IF MODE = 3 THEN
	z := 0;
	FOR n := 0 TO 4 DO (* konvertiere DWORD auf BYTE-Array *)
		FOR n1 := 0 TO 3 DO
			hash[n] := ROL(hash[n],8);
			SHA1[z] := DWORD_TO_BYTE(hash[n]);
			z := z + 1;
		END_FOR;
	END_FOR;
END_IF;

(* revision history

ks	6. dec. 2009 rev 1.0
	original version

*)

END_FUNCTION_BLOCK

// POUs/DATA_LOG/DLOG_STORE_RRD
FUNCTION_BLOCK DLOG_STORE_RRD
VAR_IN_OUT
	X : DLOG_DATA;
END_VAR
VAR_INPUT
	ENABLE : BOOL;
	TRIG_M : BOOL;
	TRIG_T : TIME;
	URL : STRING(OSCAT_BASIC.STRING_LENGTH);
	DTI : DT;
	SEP : BYTE;
	DNS_IP4 : DWORD;
	TIMEOUT : TIME;
END_VAR
VAR_OUTPUT
	ERROR_C : DWORD;
	ERROR_T : BYTE;
END_VAR
VAR
	UCB : UNI_CIRCULAR_BUFFER;
	IP_C : IP_C; (* IP_Control Verwaltungsstruktur *)
	S_BUF : NETWORK_BUFFER;
	R_BUF : NETWORK_BUFFER;
	URL_DATA : url;
	DNS_CLIENT : DNS_CLIENT;
	HTTP_GET : HTTP_GET;
	IPC : IP_CONTROL_V2;

	trig_auto : BOOL;
	trig_stored : BOOL;
	trig_tmp : BOOL;
	trig_m_last : BOOL;
	dti_last : DT := DT#2070-02-06-06:28:15;
	step_1 : INT;
	step_2 : INT;
	sep_char : STRING(1);
	url_query : STRING(OSCAT_BASIC.STRING_LENGTH);
	n : INT;

	(*
	LOG_MSG : LOG_MSG;
	_debug_enable : BOOL := TRUE;
	*)
END_VAR

(*
version 1.3		16. apr. 2012
programmer		ks
tested by			ks

DLOG_STORE_RRD der Baustein übergibt die DLOG Parameter an einen RoundRobinDatabase-Server
*)

X.DTI := DTI; (* Datum / Zeit eintragen *)
X.CLOCK_TRIG := DTI <> dti_last;
dti_last := DTI;
trig_auto := FALSE;
IF X.CLOCK_TRIG THEN (* Impuls in jeder Sekunde *)
	IF TRIG_T >= T#1000ms THEN (* automatischer Trigger *)
		trig_auto := DT_TO_UDINT(DTI) MOD (TIME_TO_UDINT(TRIG_T) / UDINT#1000) = UDINT#0;
	END_IF;
END_IF;

CASE step_1 OF

00:	IF ENABLE THEN
		X.ID_MAX := USINT#00;
		X.ADD_COM := 01; (* ADD INFO *)
		X.STORE_TYPE := BYTE#1; (* RRD-Modus *)

		ERROR_T := BYTE#0;
		ERROR_C := DWORD#0;

		X.UCB.D_MODE := 99;
		UCB(DATA:=X.UCB); (* Buffer löschen *)

		URL_DATA:=STRING_TO_URL(STR:=URL,DEFAULT_PROTOCOL:='',DEFAULT_PATH:=''); (* URL zerlegen *)
		sep_char := OSCAT_BASIC.CHR_TO_STRING(SEP);
		url_query := URL_DATA.QUERY;
		step_1 := 30;

		(* ---------------- Debug-Message -----------------------*)
		(*IF _debug_enable THEN
			LOG_CL.NEW_MSG := 'FILE_RRD1 - Start: DATE [~2]';
			LOG_CL.PRINTF[2] := DT_TO_STRING(DTI);
			LOG_MSG();
		END_IF;*)
		(* -----------------------------------------------------------------*)

	END_IF;

30:	(* LOG-Trigger verarbeiten *)
	trig_tmp := (TRIG_M AND NOT trig_m_last) OR trig_auto OR X.ADD_DATA_REQ;

	IF ENABLE = FALSE THEN (* ENABLE = 0 -> Log Stop *)
		X.ADD_COM := 00;
		step_1 := 00;

		(* ---------------- Debug-Message -----------------------*)
		(*IF _debug_enable THEN
			LOG_CL.NEW_MSG := 'FILE_RRD1 - Stop: DATE [~2]';
			LOG_CL.PRINTF[2] := DT_TO_STRING(DTI);
			LOG_MSG();
		END_IF;*)
		(* -----------------------------------------------------------------*)

	ELSIF ENABLE THEN
		IF trig_tmp OR trig_stored THEN (* manueller, automatischer oder externer Trigger *)
			trig_stored := FALSE;
			X.ADD_COM := 03; (* ADD DATA *)
			(* ---------------- Debug-Message -----------------------*)
			(*IF _debug_enable THEN
				LOG_CL.NEW_MSG := 'FILE_RRD1 - Trig: DATE [~2]';
				LOG_CL.PRINTF[2] := DT_TO_STRING(DTI);
				LOG_MSG();
			END_IF;*)
			(* -----------------------------------------------------------------*)
		ELSE
			X.ADD_COM := 04;	(* ADD DATA REQ *)
		END_IF;
	END_IF;

END_CASE;
X.ADD_DATA_REQ := FALSE; (* externe Anforderung rücksetzen *)

(* ##################################### *)

CASE step_2 OF

00:	IF X.UCB.BUF_COUNT >= USINT_TO_INT(X.ID_MAX) THEN (* genug Einträge vorhanden *)
		URL_DATA.QUERY := url_query; (* original Query wiederherstellen *)
		n := 1;
		WHILE n <= USINT_TO_INT(X.ID_MAX) DO
			X.UCB.D_MODE := 12; (* Element lesen und löschen *)
			UCB(DATA:=X.UCB);
			IF n < USINT_TO_INT(X.ID_MAX) THEN (* Trennzeichen hinzufügen *)
				X.UCB.D_STRING := CONCAT(X.UCB.D_STRING,sep_char);
			END_IF;
			IF LEN(X.UCB.D_STRING) + LEN(URL_DATA.QUERY) <= OSCAT_BASIC.STRING_LENGTH THEN
				URL_DATA.QUERY := CONCAT(URL_DATA.QUERY,X.UCB.D_STRING); (* Query mit LOG-Daten ergänzen *)
				step_2 := 40;
			ELSE
				ERROR_T := BYTE#4; (* LOG-Daten können nicht in URL gepackt werden *)
				ERROR_C := DWORD#1;
				step_2 := 100;
			END_IF;
			n := n + 1;
		END_WHILE;;
	END_IF;

40:	IF DNS_CLIENT.DONE THEN
		step_2 := 60;
	ELSIF (DNS_CLIENT.ERROR > DWORD#0) THEN
		ERROR_C := DNS_CLIENT.ERROR; (* Fehlerbehandlung *)
		ERROR_T := BYTE#1;
		step_2 := 100;
	END_IF;

60:	IF HTTP_GET.DONE THEN
		n := UINT_TO_INT(HTTP_GET.BODY_START);
		IF R_BUF.BUFFER[n] <> BYTE#48 THEN (* ASCII '0' *)
			ERROR_C := DWORD#1;
			ERROR_T := BYTE#3;
		END_IF;
		step_2 := 100;

	ELSIF HTTP_GET.ERROR > DWORD#0 THEN (* Fehlerbehandlung *)
		ERROR_C := HTTP_GET.ERROR;
		ERROR_T := BYTE#2;
		step_2 := 100;
	END_IF;

100:	IF (NOT HTTP_GET.DONE) THEN (* UNLOCK HTTP DATA *)
		step_2 := SEL(ERROR_T = BYTE#0, 120,0);
	END_IF;

120:	IF NOT ENABLE THEN
		step_2 := 0;
	END_IF;

END_CASE;

HTTP_GET(IP_C:=IP_C,S_BUF:=S_BUF,R_BUF:=R_BUF,IP4:=DNS_CLIENT.IP4,GET:=step_2=60,MODE:=2,UNLOCK_BUF:=step_2=100,URL_DATA:=URL_DATA); (* HTTP_GET *)
DNS_CLIENT(IP_C:=IP_C, S_BUF:=S_BUF, R_BUF:=R_BUF, DOMAIN:=URL_DATA.DOMAIN, IP4_DNS:= DNS_IP4, ACTIVATE:=step_2=40); (* DNS-Client *)
IPC(IP:= 0, PORT:= 0 , TIME_OUT:= TIMEOUT, IP_C:= IP_C, S_BUF:= S_BUF, R_BUF:= R_BUF); (* IP_CONTROL *)

trig_m_last := TRIG_M;

(* revision history
ks	01. jan. 2011	rev 1.0
	original version

ks	13. may. 2011	rev 1.1
	ADD_DATA_REQ hinzugefügt

ks	26. july. 2011	rev 1.2
	code optimierung D_MODE 12 und bessere fehlerauswertung

ks	16. apr. 2012	rev 1.3
	neuer überarbeiteter Code
*)

END_FUNCTION_BLOCK

// POUs/NETWORK/HTTP_GET
FUNCTION_BLOCK HTTP_GET
VAR_IN_OUT
	URL_DATA : url;
	IP_C : IP_C; (* IP_Control Verwaltungsstruktur *)
	S_BUF : NETWORK_BUFFER;
	R_BUF : NETWORK_BUFFER;
END_VAR
VAR_INPUT
	IP4 : DWORD;
	GET : BOOL;
	MODE : BYTE := BYTE#2;
	UNLOCK_BUF : BOOL;
END_VAR
VAR_OUTPUT
	HTTP_STATUS : STRING;
	HEADER_START : UINT; (* HTTP Header (Message Header) *)
	HEADER_STOP : UINT; (* HTTP Header (Message Header) *)
	BODY_START : UINT; (* Message Body *)
	BODY_STOP : UINT; (* Message Body *)
	DONE : BOOL;
	ERROR : DWORD;
END_VAR
VAR
	READ_HTTP :	READ_HTTP;
	IP_FIFO : IP_FIFO;
	ip_state : BYTE;
	ip_id : BYTE;
	get_last : BOOL;
	ip4_stored : DWORD;
	state : INT;
	i : INT;
	http_1_1_host : BOOL;
	total_size : INT;
	text : STRING(OSCAT_BASIC.STRING_LENGTH);
	delimiter2b : STRING(2);
	delimiter4b : STRING(4);
	del_end : STRING(4);
	del_pos : INT;
	idx : INT;
	rcv_timeout : BOOL;
	con_rdce : BOOL;

	(*LOG_MSG : LOG_MSG;
	_debug_enable : BOOL := TRUE;*)

END_VAR

(*

version 1.3	12. apr. 2011
programmer 	ks
tested by		ks

HTTP_GET führt eine HTTP Abfrage einer Web-Seite bei einem WEB_Server durch, und stellt die Daten ausbereitet zu verfügung
*)

CASE state OF
00:	IF GET AND NOT GET_LAST THEN (* auf positive Flanke SET warten *)
		state := 10;
		ip4_stored := IP4; (* aktuelle IP4 speichern *)
		DONE := FALSE;
		total_size := 0;
		HEADER_START := UINT#0;
		HEADER_STOP := UINT#0;
		BODY_START := UINT#0;
		BODY_STOP := UINT#0;
		HTTP_STATUS := '';
		ERROR := DWORD#0;
		ip_state := BYTE#1; (* Anmelden *)
		delimiter2b := '$0D$0A';
		delimiter4b := '$0D$0A$0D$0A';
	        	(*####################  DEBUG-MESSAGE  ###################################*)
		(*IF _debug_enable THEN
	       		LOG_CL.NEW_MSG := 'HTTP: S00 START /IP_ID ~4';
	            	LOG_CL.PRINTF[4]  := BYTE_TO_STRING(IP_ID);
	            	LOG_MSG();
	        	END_IF;*)
	        	(*########################################################################*)
	END_IF;

10:	IF ip_state = BYTE#3 THEN (* Bei IP_Control anmelden und auf freigabe warten *)
		idx := 0;
		text := CONCAT('GET ',URL_DATA.PATH);
		OSCAT_BASIC._STRING_TO_BUFFER(STR:=text,POS:=idx,PT:=ADR(S_BUF.BUFFER),SIZE:=SIZEOF(S_BUF.BUFFER)); (* GET path in buffer kopieren *)
		idx := idx + LEN(text);

		IF LEN(URL_DATA.QUERY) > 0 THEN
			S_BUF.BUFFER[idx] := 63; (* ASCII '?' *)
			idx := idx + 1;
			OSCAT_BASIC._STRING_TO_BUFFER(STR:=URL_DATA.QUERY,POS:=idx,PT:=ADR(S_BUF.BUFFER),SIZE:=SIZEOF(S_BUF.BUFFER)); (* QUERY in buffer kopieren *)
			idx := idx + LEN(URL_DATA.QUERY);
		END_IF;

		IF MODE >= BYTE#2 THEN (* gewünschte HTTP Version uebergeben *)
			text := ' HTTP/1.1';
		ELSE
			text := ' HTTP/1.0';
		END_IF;
		text := CONCAT(text,delimiter2b);
		OSCAT_BASIC._STRING_TO_BUFFER(STR:=text,POS:=idx,PT:=ADR(S_BUF.BUFFER),SIZE:=SIZEOF(S_BUF.BUFFER)); (* HTTP Version in buffer kopieren *)
		idx := idx + LEN(text);

		IF MODE = BYTE#1 THEN (* HTTP/1.0 mit persistenter Verbindung gewünscht *)
			text := CONCAT('Connection: Keep-Alive',delimiter2b); (* workaround für pcworx -> kein $0D$0A als Stringkonstante möglich *)
		ELSIF MODE = BYTE#3 THEN (* HTTP/1.1 ohne persistenter Verbindung gewünscht *)
			text := CONCAT('Connection: Close',delimiter2b); (* workaround für pcworx -> kein $0D$0A als Stringkonstante möglich *)
		ELSE
			text := '';
		END_IF;
		text := CONCAT(text,URL_DATA.HEADER);
		OSCAT_BASIC._STRING_TO_BUFFER(STR:=text,POS:=idx,PT:=ADR(S_BUF.BUFFER),SIZE:=SIZEOF(S_BUF.BUFFER)); (* HTTP Version in buffer kopieren *)
		idx := idx + LEN(text);

		text := CONCAT('Host: ',URL_DATA.DOMAIN);
		text := CONCAT(text,delimiter4b); (* workaround für pcworx -> kein $0D$0A als Stringkonstante möglich *)
		OSCAT_BASIC._STRING_TO_BUFFER(STR:=text,POS:=idx,PT:=ADR(S_BUF.BUFFER),SIZE:=SIZEOF(S_BUF.BUFFER)); (* HTTP Host in buffer kopieren *)
		idx := idx + LEN(text);

		(* IP Datenverkehr einrichten *)
		IF URL_DATA.PORT = WORD#0 THEN
			IP_C.C_PORT := WORD#80; (* Standard-Portnummer verwenden *)
		ELSE
			IP_C.C_PORT := URL_DATA.PORT; (* Portnummer aus URL verwenden *)
		END_IF;

		IP_C.C_IP := ip4_stored; (* IP eintragen *)
		IP_C.C_MODE := BYTE#0; (* Mode: TCP+AKTIV+PORT+IP *)
		IP_C.C_ENABLE := TRUE; (* Verbindungsaufbau freigeben *)
		IP_C.TIME_RESET := TRUE; (* Zeitueberwachung rücksetzen *)
		IP_C.R_OBSERVE := TRUE; (* Datenempfang ueberwachen *)
		S_BUF.SIZE := INT_TO_UINT(idx); (* Sendelänge eintragen *)
		R_BUF.SIZE := UINT#0; (* Empfangslänge rücksetzen *)

		state := 30;
	        	(*####################  DEBUG-MESSAGE  ###################################*)
	        	(*IF _debug_enable THEN
	        		LOG_CL.NEW_MSG := 'HTTP: S20 SEND /IP_ID ~4';
	            	LOG_CL.PRINTF[4]  := BYTE_TO_STRING(IP_ID);
	            	LOG_MSG();
	        	END_IF;*)
	        	(*########################################################################*)
	END_IF;

30:	rcv_timeout := (IP_C.ERROR AND DWORD#16#0000_FF00) = DWORD#16#0000_FF00;
	con_rdce :=     (IP_C.ERROR AND DWORD#16#FD00_0000) = DWORD#16#FD00_0000;

	IF S_BUF.SIZE = UINT#0 THEN
		IF total_size = 0 THEN
			IF R_BUF.SIZE > UINT#15 THEN; (* länge der empfangenen Daten prüfen *)

				(* HTTP HEADER Ende suchen -> durch $0D$A$0D$A erkennbar bei DEC RT-11,CP/M,MS-DOS,Windows *)
				del_end := '$0D$0A$0D$0A';
				del_pos := OSCAT_BASIC.BUFFER_SEARCH(PT:=ADR(R_BUF.BUFFER),SIZE:=R_BUF.SIZE,STR:=del_end,POS:=0,IGN:=FALSE);

				(* kein Ende gefunden ? -> andere Ende-Codierung suchen *)
				IF del_pos = 0 THEN
					del_end := '$0A$0A';
					(* HTTP HEADER Ende suchen -> durch $0A$0A erkennbar bei Multics, Unix-Derivate,Mac OS X *)
					del_pos := OSCAT_BASIC.BUFFER_SEARCH(PT:=ADR(R_BUF.BUFFER),SIZE:=R_BUF.SIZE,STR:=del_end,POS:=0,IGN:=FALSE);
				END_IF;

				IF del_pos > 0 THEN
					HEADER_START := UINT#0;
					HEADER_STOP := INT_TO_UINT(del_pos + LEN(del_end) - 1);
					TOTAL_SIZE := -1; (* HTTP Header empfangen aber noch keine gesamtlänge bekannt *)
				END_IF;
		                	(*####################  DEBUG-MESSAGE  ###################################*)
		                	(*IF _debug_enable THEN
		                   	LOG_CL.NEW_MSG := 'HTTP: S20 HEADER_START ~1 / HEADER_STOP ~2/IP_ID ~4';
		                   	LOG_CL.PRINTF[4]  := BYTE_TO_STRING(IP_ID);
		                   	LOG_CL.PRINTF[1]  := UINT_TO_STRING(HEADER_START);
		                   	LOG_CL.PRINTF[2]  := UINT_TO_STRING(HEADER_STOP);
		                   	LOG_MSG();
		                	END_IF;*)
		                	(*########################################################################*)

				(* HTTP Statuscode auswerten: (kann 1.0 oder 1.1 sein *)
				READ_HTTP(size:=HEADER_STOP,pos:=0,SRC:='',pt:=R_BUF.BUFFER);

				i := LEN(READ_HTTP.READ_HTTP);
				IF i > 7 THEN
					(* HTTP Version von HOST auswerten 1.0 oder 1.1 *)
					text:=MID(READ_HTTP.READ_HTTP,1,3);
					http_1_1_host := text = '1';

					(* Code und Meldung isolieren *)
					HTTP_STATUS := RIGHT(READ_HTTP.READ_HTTP,i-4);
				END_IF;

				(* positive HTTP Anfrage ? *)
				IF FIND(HTTP_STATUS,'200') > 0 THEN

					(* 'Content-Length: Wert einlesen auswerten *)
					READ_HTTP(size:=HEADER_STOP,pos:=0,SRC:='CONTENT-LENGTH',pt:=R_BUF.BUFFER);
					text:=READ_HTTP.READ_HTTP;

					IF LEN(text) >= 1 THEN
						IF OSCAT_BASIC.IS_NUM(str:=text) THEN
							(* erwartete gesamtmenge an Bytes berechnen *)
							total_size := STRING_TO_INT(text) + UINT_TO_INT(HEADER_STOP) + 1;
                           					(*####################  DEBUG-MESSAGE  ###################################*)
                           					(*IF _debug_enable THEN
                              					LOG_CL.NEW_MSG := 'HTTP: S20 HEADER ~1, BODY ~2 TOTAL ~3 /IP_ID ~4';
                             					LOG_CL.PRINTF[4]  := BYTE_TO_STRING(IP_ID);
                               					LOG_CL.PRINTF[1]  := UINT_TO_STRING(HEADER_STOP);
                               					LOG_CL.PRINTF[2]  := INT_TO_STRING(TOTAL_SIZE-UINT_TO_INT(HEADER_STOP));
                               					LOG_CL.PRINTF[3]  := INT_TO_STRING(TOTAL_SIZE);
                              					LOG_MSG();
                          					END_IF;*)
                          					(*########################################################################*)
						END_IF;
					END_IF;
				ELSE
					ERROR := DWORD#16#000000FC; (* Fehler durch HTTP-Statuscodes *)
				END_IF;
			END_IF;
		(* 1. bei bekannter Content-Length wird nach erhalt der erwartenen Daten die verbindung beendet *)
		(* 2. bei persistenter Verbindung muss bei unbekannter Datenmenge auf Receive-Timeout gewartet werden *)
		(* 3. wenn nach datenempfang die verbindung vom host unterbrochen wird *)
		ELSIF (R_BUF.SIZE >= INT_TO_UINT(total_size)) OR
			(R_BUF.SIZE > UINT#0 AND total_size < 0 AND ((rcv_timeout OR con_rdce) OR (IP_C.C_STATE = BYTE#1))) THEN

			IF R_BUF.SIZE - 1 > HEADER_STOP THEN (* BODY Daten vorhanden *)
				BODY_START := HEADER_STOP + UINT#1;
				BODY_STOP := R_BUF.SIZE - 1;
		                	(*####################  DEBUG-MESSAGE  ###################################*)
		                	(*IF _debug_enable THEN
		                   	LOG_CL.NEW_MSG := 'HTTP: S20 BODY ~1, START ~2 END ~3 /IP_ID ~4';
		                   	LOG_CL.PRINTF[4]  := BYTE_TO_STRING(IP_ID);
		                   	LOG_CL.PRINTF[1]  := UINT_TO_STRING(HEADER_STOP);
		                   	LOG_CL.PRINTF[2]  := UINT_TO_STRING(BODY_START);
		                   	LOG_CL.PRINTF[3]  := UINT_TO_STRING(BODY_STOP);
		                   	LOG_MSG();
		               	END_IF;*)
		               	(*########################################################################*)
			END_IF;

			DONE := TRUE;
			IP_C.C_ENABLE := FALSE; (* Verbindung abbauen *)
			state := 40;
            		(*####################  DEBUG-MESSAGE  ###################################*)
            		(*IF _debug_enable THEN
                			LOG_CL.NEW_MSG := 'HTTP: S30 OK /IP_ID ~4';
                			LOG_CL.PRINTF[4]  := BYTE_TO_STRING(IP_ID);
                			LOG_MSG();
            		END_IF;*)
            		(*########################################################################*)
		END_IF;
	END_IF;

	IF IP_C.ERROR <> DWORD#0 THEN
		(* bei unbekannter Content-size ist nicht bekannt ob bzw wieviele Telegramme noch folgen werden *)
		(* darum wird nach receive-timeout oder Remote disconnect error der fehler wieder ausgefiltert (logischer fehler) *)
		IF rcv_timeout AND DONE THEN
			IP_C.ERROR := IP_C.ERROR AND DWORD#16#FFFF_00FF; (* Fehler wieder rücksetzen *)
		ELSIF con_rdce AND DONE THEN
			IP_C.ERROR := IP_C.ERROR AND DWORD#16#00FF_FFFF; (* Fehler wieder rücksetzen *)
		ELSE
			ERROR := IP_C.ERROR;
		END_IF;
	END_IF;

	IF ERROR > DWORD#0 THEN
		IP_C.C_ENABLE := FALSE; (* Verbindungsaufbau sperren *)
		state := 40;
	        	(*####################  DEBUG-MESSAGE  ###################################*)
	        	(*IF _debug_enable THEN
	            	LOG_CL.NEW_MSG := 'HTTP: S30 ERROR ~1 /IP_ID ~4';
	            	LOG_CL.PRINTF[1]  := DWORD_TO_STRING(ERROR);
	            	LOG_CL.PRINTF[4]  := BYTE_TO_STRING(IP_ID);
	            	LOG_MSG();
	        	END_IF;*)
	        	(*########################################################################*)
	END_IF;

40:	IF (UNLOCK_BUF OR NOT DONE) THEN (* Warten auf Release und Verbindung beendet -> IP_ID vom Stack nehmen *)
		IP_STATE := BYTE#4; (* Abmelden *)
		DONE := FALSE;
		state := 0;
	END_IF;
END_CASE;

get_last := GET; (* letzten Status sichern zur Flankenerkennung *)

IP_FIFO(FIFO:=IP_C.FIFO,STATE:=ip_state,ID:=ip_id); (* IP_FIFO *)

(* revision history
ks	18. oct. 2008	rev 1.0
	original version

ks	20. oct. 2009	rev 1.1
	Fehler bei body-suche bei $0a$0a korrigiert,Codeoptimierung,
	new VAR del_pos , del_end (Networkbuffer und Buffer-funktionen auf Basis 0)

ks	28. oct. 2009	rev 1.2
	über url.header können zusätzliche header-infos übergeben werden

ks	12. apr. 2011	rev 1.3
	verbesserte fehlererkennung und fehlerkorrektur bei buffer_to_string
*)

END_FUNCTION_BLOCK

// POUs/NETWORK/READ_HTTP
FUNCTION_BLOCK READ_HTTP
VAR_INPUT
	SIZE : UINT;
	POS : INT;
	SRC : STRING;
END_VAR
VAR_IN_OUT
	PT : NW_BUF_LONG;
END_VAR
VAR_OUTPUT
	READ_HTTP : STRING(OSCAT_BASIC.STRING_LENGTH);
END_VAR
VAR
	index : INT;
	s1 : INT;
	e1 : INT;
	stop : INT;
END_VAR

(*

version 1.1 20. oct. 2009
programmer 	ks
tested by	ks

READ_HTTP wertet die Informationen einer HTTP-Request aus, und stellt die Daten zu Verfügung.
*)

stop := UINT_TO_INT(SIZE) - 1;

IF LEN(SRC) = 0 THEN
	(* wenn kein Suchbegriff vorhanden ist, dann den HTTP-STATUS auswerten *)
	SRC := 'HTTP/'; (* neuer Suchbegriff *)
ELSE
	(* gesuchten Parametertext ergänzen *)
	SRC := CONCAT(SRC,': ');
END_IF;

s1 := OSCAT_BASIC.BUFFER_SEARCH(pt:=ADR(PT),SIZE:=SIZE,STR:=SRC,POS:=POS,IGN:=TRUE);

IF s1 >= 0 THEN (* Text found *)
	e1 := s1;

	(* search start of line *)
	index := s1 - 1;
	WHILE (index > 0) DO
		IF pt[index] < BYTE#32 THEN EXIT; END_IF;
		s1 := s1 - 1;
		index := index - 1;
	END_WHILE;

	(* search end of line *)
	index := e1 + 1;
	WHILE (index <= stop) DO
		IF pt[index] < BYTE#32 THEN EXIT; END_IF;
		e1 := e1 + 1;
		index := index + 1;
	END_WHILE;

	s1 := s1 + LEN(SRC); (* 'suchbegriff: ' nicht mitkopieren *)

	(* copy string *)
	READ_HTTP := OSCAT_BASIC.BUFFER_TO_STRING(PT:=ADR(PT),SIZE:=SIZE,START:=s1,STOP:=e1);
ELSE
	READ_HTTP := '';
END_IF;

(* revision history

ks	18. oct. 2008	rev 1.0
	original version

ks	20. oct. 2009	rev 1.1
	Networkbuffer und Buffer-funktionen auf Basis 0

*)

END_FUNCTION_BLOCK

// POUs/DATA_LOG/DLOG_STRING
FUNCTION_BLOCK DLOG_STRING
VAR_IN_OUT
	X : DLOG_DATA;
END_VAR
VAR_INPUT
	STR : STRING;
	COLUMN : STRING(40);
END_VAR
VAR_OUTPUT
END_VAR
VAR
	UCB : UNI_CIRCULAR_BUFFER;
	id : WORD;
	str_last : STRING;
END_VAR

(*
version 1.3		19. apr. 2012
programmer		ks
tested by		ks

DLOG_STRING legt den STRING im FIFO-RING-Buffer ab um diesen mit den Baustein DLOG_STORE_*  aufzuzeichnen
*)

CASE x.ADD_COM OF

01:	(* ADD INFO *)
	X.ID_MAX := X.ID_MAX + USINT#1;
	id := WORD#16#0101; (* Quelltype STRING , Zieltype STRING *)
02:	(* ADD HEADER *)
	X.UCB.D_STRING := COLUMN;
	X.UCB.D_HEAD := id;
	X.UCB.D_MODE := 1;
	UCB(DATA:=X.UCB); (* Daten eintragen *)
03:	(* ADD DATA *)
	X.UCB.D_STRING := str_last;
	X.UCB.D_HEAD := id;
	X.UCB.D_MODE := 1;
	UCB(DATA:=X.UCB); (* Daten eintragen *)
END_CASE;
str_last := STR;

(* revision history
ks	01. jan. 2011	rev 1.0
	original version

ks	17. may. 2011	rev 1.1
	COLUMN STRING(40)

ks	25. july.   2011	rev 1.2
	neue head information

ks	19. apr.   2012	rev 1.3
	code neu überarbeitet
*)

END_FUNCTION_BLOCK

// POUs/NETWORK/DNS_DYN
FUNCTION_BLOCK DNS_DYN
VAR_IN_OUT
	IP_C : IP_C; (* IP_Control Verwaltungsstruktur *)
	S_BUF : NETWORK_BUFFER;
	R_BUF : NETWORK_BUFFER;
END_VAR
VAR_INPUT
	ENABLE : BOOL;
	UPDATE : BOOL;
	T_UPDATE : TIME := T#1h;
	MODE : BYTE;
	HOSTNAME : STRING(30);
	USERNAME : STRING(20);
	PASSWORD : STRING(20);
	IP4 : DWORD;
END_VAR
VAR_OUTPUT
	BUSY : BOOL;
	DONE : BOOL;
	ERROR_C : DWORD;
	ERROR_T : BYTE;
END_VAR
VAR
	DNS_CLIENT : DNS_CLIENT;
	HTTP_GET : HTTP_GET;
	BASE64_ENCODE_STR : BASE64_ENCODE_STR;
	URL_DATA : url;
	update_last : BOOL;
	state : INT;
	base64_done : BOOL;
	s1 : STRING(144);
	s2 : STRING(192);
	w : TON;
END_VAR

(*

version 1.2		02. dec. 2009
programmer 		ks
tested by		ks

YAHOO_WEATHER lädt vom Yahoo-Webserver einen Wetter RSS-Feed und analysiert die Daten und legt diese in einem Array ab
*)

CASE state OF

00:	IF ENABLE AND ((UPDATE AND NOT update_last) OR w.Q) THEN
		state := 20;
		DONE := FALSE;
		BUSY := TRUE;
		ERROR_C := DWORD#0;
		ERROR_T := BYTE#0;

		IF MODE = 0 THEN (* dyndns.org *)
			s2 := CONCAT('http://members.dyndns.org/nic/update?hostname=',HOSTNAME);
		ELSE (* selfhost.de *)
			s2 := 'http://carol.selfhost.de/nic/update?hostname=1';
		END_IF;
		IF IP4 > 0 THEN (* parametrierte IP verwenden *)
			s1 := CONCAT('&myip=',IP4_TO_STRING(IP4));
			s2 := CONCAT(s2,s1);
		END_IF;
		URL_DATA:=STRING_TO_URL(STR:=s2, DEFAULT_PROTOCOL:='', DEFAULT_PATH:=''); (* URL for DNS UND HTTP-GET *)
		s1 := CONCAT(USERNAME,':');
		s1 := CONCAT(s1,PASSWORD); (* BASE64 Encode Text *)
	END_IF;

20:	IF DNS_CLIENT.DONE THEN (* DNS_CLIENT *)
			state := 40;
	ELSIF (DNS_CLIENT.ERROR > DWORD#00) THEN (* Fehlerbehandlung *)
		ERROR_C := DNS_CLIENT.ERROR;
		ERROR_T := BYTE#01;
		BUSY := FALSE;
		state := 0;
	END_IF;

40: IF base64_done THEN (* BASE64 Encode beendet ? *)
		s1 := CONCAT('Authorization: Basic ',s2);
		s1 := CONCAT(s1,'$0D$0AUser-Agent: x$0D$0A');
		URL_DATA.HEADER := s1;
		state := 60;
	END_IF;

60:	IF HTTP_GET.DONE THEN
		state := 0;
		BUSY := FALSE;
		DONE := TRUE;

		(* !! Codes !!
		Successful Updates: 		good , nchg
		Update Syntax Errors:		badsys , badagent
		Account-Related Errors:		badauth , !donator
		Hostname-Related Errors:	notfqdn , nohost , !yours , numhost , abuse
		Server Error Conditions:	dnserr , 911
		*)
		s2 := OSCAT_BASIC.BUFFER_TO_STRING(PT:=ADR(R_BUF.BUFFER),SIZE:=SIZEOF(R_BUF.BUFFER),START:=HTTP_GET.BODY_START + 3,STOP:=HTTP_GET.BODY_STOP - 7);
		IF FIND(s2,'good') = 0 THEN
			IF FIND(s2,'nochg') = 0 THEN
				ERROR_C := DWORD#1;
				ERROR_T := BYTE#03;
				DONE := FALSE;
			END_IF;
		END_IF;
	ELSIF (HTTP_GET.ERROR > DWORD#00) THEN (* Fehlerbehandlung *)
		ERROR_C := HTTP_GET.ERROR;
		ERROR_T := BYTE#02;
		BUSY := FALSE;
		state := 0;
	END_IF;

END_CASE;

DNS_CLIENT(IP_C:=IP_C,	S_BUF:=S_BUF, R_BUF:=R_BUF,DOMAIN:=URL_DATA.DOMAIN, IP4_DNS:=0, ACTIVATE:=state=20); (* DNS_CLIENT *)
HTTP_GET( IP_C:=IP_C, S_BUF:=S_BUF, R_BUF:=R_BUF, IP4:=DNS_CLIENT.IP4, GET:=state=60, MODE:=2, UNLOCK_BUF:=state<>60,URL_DATA:=URL_DATA); (* HTTP_GET *)
BASE64_ENCODE_STR( RUN:=state=40, STR1:=s1, STR2:=s2, DONE=>base64_done); (* BASE64 Encode *)

IF T_UPDATE > T#0ms THEN w(IN:=state=0, PT:=T_UPDATE); END_IF;
update_last := UPDATE;

(* revision history
ks	01. jan. 2010	rev 1.0
	original version

*)

END_FUNCTION_BLOCK

// POUs/WEATHER/YAHOO_WEATHER
FUNCTION_BLOCK YAHOO_WEATHER
VAR_IN_OUT
	IP_C : IP_C; (* IP_Control Verwaltungsstruktur *)
	S_BUF : NETWORK_BUFFER;
	R_BUF : NETWORK_BUFFER;
	YW : YAHOO_WEATHER_DATA;
END_VAR
VAR_INPUT
	ACTIVATE : BOOL;
	UNITS : BOOL;
	LOCATION : STRING(20);
END_VAR
VAR_OUTPUT
	BUSY : BOOL;
	DONE : BOOL;
	ERROR_C : DWORD;
	ERROR_T : BYTE;
END_VAR
VAR
	CTRL : XML_CONTROL;
	XML_READER : XML_READER;
	URL_DATA : url;
	DNS_CLIENT : DNS_CLIENT;
	HTTP_GET : HTTP_GET;
	last_state : BOOL;
	value_int : INT;
	value_real : REAL;
	v_real : REAL;
	state : INT;
END_VAR

(*

version 1.3		04. may. 2011
programmer 		ks
tested by			ks

YAHOO_WEATHER lädt vom Yahoo-Webserver einen Wetter RSS-Feed und analysiert die Daten und legt diese in einem Array ab
*)

CASE state OF

00:	IF ACTIVATE AND NOT last_state THEN
		state := 20;
		DONE := FALSE;
		BUSY := TRUE;
		ERROR_C := DWORD#0;
		ERROR_T := BYTE#0;
	END_IF;

20: (* URL for DNS UND HTTP-GET *)
	(* Example: http://weather.yahooapis.com/forecastrss?p=94089&u=c *)
	URL_DATA:=STRING_TO_URL(STR:='http://weather.yahooapis.com/forecastrss',
							DEFAULT_PROTOCOL:='',
							DEFAULT_PATH:=''
							);
  	URL_DATA.QUERY := CONCAT('w=',LOCATION);

	IF UNITS THEN
		URL_DATA.QUERY := CONCAT(URL_DATA.QUERY,'&u=f'); (* fahrenheit *)
	ELSE
		URL_DATA.QUERY := CONCAT(URL_DATA.QUERY,'&u=c'); (* celsius *)
	END_IF;
	state := 40;

40:	IF DNS_CLIENT.DONE THEN
		state := 60;
	ELSIF (DNS_CLIENT.ERROR > DWORD#00) THEN
		(* Fehlerbehandlung *)
		ERROR_C := DNS_CLIENT.ERROR;
	ERROR_T := BYTE#01;
		state   := 100;
	END_IF;

60:	IF HTTP_GET.DONE THEN
		state := 80;
		CTRL.START_POS := HTTP_GET.BODY_START;
		CTRL.STOP_POS := HTTP_GET.BODY_STOP;
		CTRL.COMMAND := WORD#2#10000000_00011000; (* ONLY TEXT AND ATTRIBUTE *)
		CTRL.WATCHDOG  := T#1ms;

	ELSIF (HTTP_GET.ERROR > DWORD#00) THEN
		(* Fehlerbehandlung *)
		ERROR_C := HTTP_GET.ERROR;
		ERROR_T := BYTE#02;
		state := 100;
	END_IF;

80: XML_READER(CTRL:=CTRL,BUF:=R_BUF.BUFFER); (* XML Daten seriell lesen *)
	IF CTRL.TYP < 98 THEN (* nur auswerten wenn kein Watchdog durchlauf *)
		value_int := 0;
		value_real := 0.0;
		(* automatische konvertierung in real und int ausführen *)
		IF LEN(CTRL.VALUE) <= 20 THEN
			v_real:=OSCAT_BASIC.FLOAT_TO_REAL(FLT:=CTRL.VALUE);
			IF OSCAT_BASIC.CHK_REAL(v_real) = 0 THEN (* !!! prüft auf gültigen REAL Wert, ansonsten stürzt Twincat ab !!!!  *)
				value_real := v_real;
				value_int := REAL_TO_INT(value_real);
			END_IF;
		END_IF;

		IF CTRL.COUNT < UINT#52 THEN (* Performance-Teilung *)
			(* ------------ Teil 1 --------------*)
			CASE UINT_TO_INT(CTRL.COUNT) OF
			027: YW.TimeToLive := value_int;
			030: YW.location_city := CTRL.VALUE;
			031: YW.location_region := CTRL.VALUE;
			032: YW.location_country := CTRL.VALUE;
			035: YW.unit_temperature := CTRL.VALUE;
			036: YW.unit_distance := CTRL.VALUE;
			037: YW.unit_pressure := CTRL.VALUE;
			038: YW.unit_speed := CTRL.VALUE;
			041: YW.wind_chill := value_int;
			042: YW.wind_direction := value_int;
			043: YW.wind_speed := value_real;
			046: YW.atmosphere_humidity := value_int;
			047: YW.atmosphere_visibility := value_real;
			048: YW.atmosphere_pressure := value_int;
			049: YW.atmosphere_rising := value_int;
			END_CASE;
		ELSE
			(* ------------ Teil 2 --------------*)
			CASE UINT_TO_INT(CTRL.COUNT) OF
			052: YW.astronomy_sunrise := CTRL.VALUE;
			053: YW.astronomy_sunset := CTRL.VALUE;
			077: YW.geo_latitude := value_real;
			080: YW.geo_longitude := value_real;
			089: YW.cur_conditions_text := CTRL.VALUE;
			090: YW.cur_conditions_code := value_int;
				YW.cur_conditions_icon := value_int;
			091: YW.cur_conditions_temp := value_int;
			100: YW.forcast_today_low_temp := value_int;
			101: YW.forcast_today_high_temp := value_int;
			102: YW.forcast_today_text := CTRL.VALUE;
			103: YW.forcast_today_code := value_int;
				YW.forcast_today_icon := value_int;
			108: YW.forcast_tomorrow_low_temp := value_int;
			109: YW.forcast_tomorrow_high_temp := value_int;
			110: YW.forcast_tomorrow_text := CTRL.VALUE;
			111: YW.forcast_tomorrow_code := value_int;
				YW.forcast_tomorrow_icon := value_int;
			END_CASE;
		END_IF;
	ELSIF CTRL.TYP = 99 THEN (* EXIT - letztes Element gelesen *)
		DONE  := TRUE;
		state := 100;
	END_IF; 

100:
	(* UNLOCK HTTP DATA *)
	IF (NOT HTTP_GET.DONE) THEN
		state := 0;
		BUSY := FALSE;
		DONE := ERROR_T = BYTE#0;
	END_IF; 

	END_CASE;

(* ---------------- DNS --------------- *)
DNS_CLIENT(	IP_C:=IP_C,
			S_BUF:=S_BUF,
			R_BUF:=R_BUF,
			DOMAIN:=URL_DATA.DOMAIN,
			IP4_DNS:=DWORD#00,
			ACTIVATE:=state=40 (* DNS Start *)
			);
(* nicht oder nicht direkt verwendete Parameter *)
(*	DWORD :=DNS_CLIENT.IP4;
	BOOL  :=DNS_CLIENT.DONE;
	BYTE  :=DNS_CLIENT.ERROR; *)
(* -------------------------------------*)

(* ------------- HTTP_GET --------------- *)
HTTP_GET(	IP_C:=IP_C,
			S_BUF:=S_BUF,
			R_BUF:=R_BUF,
			IP4:=DNS_CLIENT.IP4,
			GET:=state=60,
			MODE:=BYTE#2, (* HTTP 1.1 mit persistenter Verbindung *)
			UNLOCK_BUF:=state=100,
			URL_DATA:=URL_DATA
			);

(* nicht oder nicht direkt verwendete Parameter *)
(*	STRING := HTTP_GET.HTTP_STATUS;
	UINT :=HTTP_GET.HEADER_START;
	UINT :=HTTP_GET.HEADER_STOP;
	UINT :=HTTP_GET.BODY_START;
	UINT :=HTTP_GET.BODY_STOP;
	BOOL :=HTTP_GET.DONE;
	BYTE :=HTTP_GET.ERROR;
*)
(* -------------------------------------*)

last_state := ACTIVATE;

(* revision history
ks	18. dez. 2008	rev 1.0
	original version

ks	01. oct. 2009	rev 1.1
	YAHOO_WEATHER_DATA

ks	24. sep. 2010	rev 1.2
	new URL-Location-parameter and REAL_CHECK (TwinCat BUG) 

ks	04. may. 2011	rev 1.3
	neue elemente:  CUR_CONDITIONS_ICON, FORCAST_TODAY_ICON, FORCAST_TOMORROW_ICON

*)

END_FUNCTION_BLOCK

// POUs/NETWORK/XML_READER
FUNCTION_BLOCK XML_READER
VAR_IN_OUT
	CTRL : XML_CONTROL;
	BUF : NW_BUF_LONG;
END_VAR
VAR
	index :	INT;
	index2 : INT;
	stop : INT;
	mode : INT;
	command : WORD;
	c :	BYTE;
	s1 : INT;
	e1 : INT;
	path_overflow : BOOL;
	empty_tag : BOOL;
	s_code : STRING(10);
	e_code : STRING(10);
	watchdog : TON;

	(*LOG_MSG : LOG_MSG;
	_debug_enable : BOOL := TRUE;*)

END_VAR

(*

version 1.2		10. mai 2010
programmer 	ks
tested by		ks

XML_READER ermöglicht das serielle Parsen und die Auswertung von XML_Elementen in einem Buffer
*)

(*

TYP
00 = UNBEKANNT
01 = ELEMENT (STANDARD)
02 = CLOSE ELEMENT 
03 = TEXT
04 = ATTRIBUTE
05 = ELEMENT (PROCESSING INSTRUCTION) 

12 = !CDATA
13 = !COMMENT
14 = !DTD ELEMENT (Document Type Declarations )

98 = WATCHDOG
99 = ENDE

Bei Typ 02 werden keine Blockdaten ausgegeben !

*)

(* ---------- Init -------------- *)
IF OSCAT_BASIC.BIT_OF_DWORD(WORD_TO_DWORD(CTRL.COMMAND),15) THEN
	COMMAND := CTRL.COMMAND;
	CTRL.COMMAND := WORD#0;

	index := UINT_TO_INT(CTRL.START_POS);
	stop := UINT_TO_INT(CTRL.STOP_POS);
	mode := 100;
	path_overflow := FALSE;

	CTRL.TYP := 0;
	CTRL.COUNT := UINT#00;
	CTRL.LEVEL := UINT#00;
	CTRL.ATTRIBUTE := '';
	CTRL.ELEMENT := '';
	CTRL.PATH := '';
	CTRL.VALUE := '';

	WATCHDOG.PT := CTRL.WATCHDOG;
END_IF;

(*----------------------------------------------- *)

IF index < 0 THEN RETURN;END_IF;

CTRL.BLOCK1_START := UINT#0;
CTRL.BLOCK1_STOP := UINT#0;
CTRL.BLOCK2_START := UINT#0;
CTRL.BLOCK2_STOP := UINT#0;

WATCHDOG(IN:=FALSE); (* Timer stoppen *)

WHILE (TRUE) DO

	(* -------------- WATCHDOG ------------------ *)
	WATCHDOG(IN:=CTRL.WATCHDOG > T#0s);
	IF WATCHDOG.Q THEN
		CTRL.TYP := 98;
    		(*####################  DEBUG-MESSAGE  ###################################*)
    		(*IF _debug_enable THEN
      			LOG_CL.NEW_MSG := 'WATCHDOG:';
      			LOG_MSG();
    		END_IF;*)
    		(*########################################################################*)
		RETURN;
	END_IF;

	(* -------------- PARSING END ------------------ *)
	IF index > stop THEN
		CTRL.COUNT := CTRL.COUNT + UINT#1;
		CTRL.TYP := 99;
    		(*####################  DEBUG-MESSAGE  ###################################*)
    		(*IF _debug_enable THEN
      			LOG_CL.NEW_MSG := 'EX: #T:~1 #C:~2 #P:~6 #L:~7';
      			LOG_CL.PRINTF[1] := INT_TO_STRING(CTRL.TYP);
      			LOG_CL.PRINTF[2] := UINT_TO_STRING(CTRL.COUNT);
      			LOG_CL.PRINTF[6] := CTRL.PATH;
      			LOG_CL.PRINTF[7] := UINT_TO_STRING(CTRL.LEVEL);
      			LOG_MSG();
    		END_IF;*)
    		(*########################################################################*)
		mode  := 0; (* Schritt ruecksetzen *)
		index := 0; (* Abarbeitung stoppen *)
		RETURN;
	END_IF;

	CASE mode OF

	100: (* ---------- ELEMENT SECTION ------------------ *)
		(* search begin of element *)
		s1 := 0;
		e1 := 0;
		WHILE (index <= stop) DO
			IF BUF[INDEX]=BYTE#60 THEN (* '<' TagBegin *)
				index := index + 1;
				C := BUF[index];
				IF C = BYTE#47 THEN (* '/' TagTerm *)
					mode := 300; (* End Element Section *)
				ELSIF C = BYTE#33 THEN (* '!' for Special Section *)
					index := index + 1;
					mode := 500;
				ELSE
					s1 := index;
				END_IF;
				EXIT;
			END_IF;
			index := index + 1;
		END_WHILE;

		(* analyse element *)
		CTRL.TYP := 0; (* TYP löschen *)
		IF s1 > 0 THEN
			WHILE (index <= stop AND e1 = 0) DO
				c := BUF[index];
				(* whitespace zeichen = Element with Attributes *)
				IF c <= BYTE#32 THEN
					(* suche nächstes druckbares zeichen *)
					index2 := index;
					WHILE (index2 <= stop) AND (BUF[index2] <= BYTE#32) DO
						index2 := index2 + 1;
					END_WHILE;
					IF BUF[index2] = BYTE#47 THEN (* pruefe auf leeres Element '/' *)
						index := index2;
						e1 := index - 2;
						CTRL.TYP := 1; (* struktur-element *)
						mode := 300;   (* Close Element *)
						EXIT;
					END_IF;

					e1 := index - 1;
					CTRL.TYP := 1; (* Element mit Attribute *)
					mode := 400;

				ELSIF c = BYTE#62 THEN (* '>' TagEnd *)

					(* pruefe auf leeres Element <xx/> *)
					index2 := index - 1;
					IF BUF[index2] = BYTE#47 THEN (* TagTerm '/' *)
						e1 := index2 - 1;
						CTRL.TYP := 1;
						EMPTY_TAG := TRUE; (* EMPTY TAG Mode *)
						mode := 200; (* TEXT Element *)
						EXIT;
					END_IF;

					e1 := index - 1;
					index2 := index + 1;

					(* untersuche nachfolgendes Element *)
					WHILE (index2 <= stop) DO
						c := BUF[index2];
						IF c = BYTE#60 THEN (* '<' TagBegin *)

							index2 := index2 + 1; (* geht bei PCWORX leider nicht anders !*)
							c := BUF[index2];
							index2 := index2 - 1;
							IF c = BYTE#47 THEN (* TagTerm '/' *)
								empty_tag := TRUE;
								mode := 200; (* TEXT Element *)
							ELSE
								mode := 100; (* Element *)
							END_IF;
							CTRL.TYP := 1; (* struktur-element *)
							EXIT;
						ELSIF c > BYTE#32  THEN (* Printable-Character *)
							CTRL.TYP := 1; (* element with text *)
							mode := 200;
							EXIT;
						END_IF;
						index2 := index2 + 1;
					END_WHILE;
				END_IF;
				index := index + 1;
			END_WHILE;
		END_IF;

		(* Neues Element gefunden*)
		IF CTRL.TYP > 0 THEN

			(* Sonderprüfung auf Processing Instruction (PI) *)
			IF BUF[s1] = BYTE#63 THEN (* '?' for Processing Instruction *)
				s1 := s1 + 1; (* führendes '?' auslassen *)
				CTRL.TYP := 5;
			END_IF;
			CTRL.BLOCK1_START := INT_TO_UINT(s1);
			CTRL.BLOCK1_STOP  := INT_TO_UINT(e1);
			CTRL.ELEMENT := OSCAT_BASIC.BUFFER_TO_STRING(PT:=ADR(BUF),SIZE:=INT_TO_UINT(stop + 1),START:=CTRL.BLOCK1_START,STOP:=CTRL.BLOCK1_STOP);
			CTRL.COUNT := CTRL.COUNT + UINT#1;
			CTRL.LEVEL := CTRL.LEVEL + UINT#1;

			IF path_overflow = FALSE THEN
				(* Stringlänge überwachen *)
				IF LEN(CTRL.PATH) + LEN(CTRL.ELEMENT) + 1 > 250 THEN
					path_overflow := TRUE;
					CTRL.PATH := 'OVERFLOW';
				ELSE
					CTRL.PATH := CONCAT(CTRL.PATH,'/');
					CTRL.PATH  := CONCAT(CTRL.PATH,CTRL.ELEMENT);
				END_IF;
			END_IF;

			IF OSCAT_BASIC.BIT_OF_DWORD(WORD_TO_DWORD(COMMAND),CTRL.TYP) THEN
        				(*####################  DEBUG-MESSAGE  ###################################*)
        				(*IF _debug_enable THEN
          				LOG_CL.NEW_MSG := 'EL: #T:~1 #C:~2 #E:~3 #P:~6 #L:~7';
          				LOG_CL.PRINTF[1] := INT_TO_STRING(CTRL.TYP);
          				LOG_CL.PRINTF[2] := UINT_TO_STRING(CTRL.COUNT);
          				LOG_CL.PRINTF[3] := CTRL.ELEMENT;
          				LOG_CL.PRINTF[6] := CTRL.PATH;
          				LOG_CL.PRINTF[7] := UINT_TO_STRING(CTRL.LEVEL);
          				LOG_MSG();
        				END_IF;*)
        				(*########################################################################*)
				RETURN;
			END_IF;
		END_IF;

	200: (* ---------- TEXT SECTION ------------------ *)
		CTRL.VALUE := '';
		IF empty_tag = FALSE THEN
			s1 := index;
			(* suche '<' EndTag*)
			WHILE (index <= stop) AND (BUF[index] <> BYTE#60) DO
				index := index + 1;
			END_WHILE;

			E1 := index - 1;
			CTRL.BLOCK1_START := INT_TO_UINT(s1);
			CTRL.BLOCK1_STOP  := INT_TO_UINT(e1);
			CTRL.VALUE := OSCAT_BASIC.BUFFER_TO_STRING(PT:=ADR(BUF),SIZE:=INT_TO_UINT(stop + 1),START:=CTRL.BLOCK1_START,STOP:=CTRL.BLOCK1_STOP);
		END_IF;

		empty_tag := FALSE;
		mode := 300; (* -> NEXT-JOB: END ELEMENT *)
		CTRL.COUNT := CTRL.COUNT + UINT#1;
		CTRL.TYP := 3;

		IF OSCAT_BASIC.BIT_OF_DWORD(WORD_TO_DWORD(command),CTRL.TYP) THEN
      			(*####################  DEBUG-MESSAGE  ###################################*)
      			(*IF _debug_enable THEN
        				LOG_CL.NEW_MSG := 'TE: #T:~1 #C:~2 #E:~3 #V:~4 #P:~6 #L:~7';
        				LOG_CL.PRINTF[1] := INT_TO_STRING(CTRL.TYP);
        				LOG_CL.PRINTF[2] := UINT_TO_STRING(CTRL.COUNT);
        				LOG_CL.PRINTF[3] := CTRL.ELEMENT;
        				LOG_CL.PRINTF[4] := CTRL.VALUE;
        				LOG_CL.PRINTF[6] := CTRL.PATH;
        				LOG_CL.PRINTF[7] := UINT_TO_STRING(CTRL.LEVEL);
        				LOG_MSG();
      			END_IF;*)
      			(*########################################################################*)
			RETURN;
		END_IF;

	300: (* ---------- END ELEMENT SECTION ------------------ *)
		WHILE (index <= stop) DO
			c := BUF[index];
			IF c = BYTE#62 THEN (* '>' TagEnd *)
				index := index + 1;
				s1 := OSCAT_BASIC.FINDB(str1:=CTRL.PATH,str2:='/');
				IF path_overflow = FALSE THEN
					IF s1 > 1 THEN
						CTRL.ELEMENT := RIGHT(CTRL.PATH,LEN(CTRL.PATH) - s1);
						CTRL.PATH := LEFT(CTRL.PATH,s1 - 1);
					ELSE
						CTRL.ELEMENT := RIGHT(CTRL.PATH,LEN(CTRL.PATH) - 1);
						CTRL.PATH :='';
					END_IF;
				END_IF;

				CTRL.LEVEL := CTRL.LEVEL - UINT#1;
				CTRL.COUNT := CTRL.COUNT + UINT#1;
				CTRL.TYP := 2;
				mode := 100;

				IF OSCAT_BASIC.BIT_OF_DWORD(WORD_TO_DWORD(COMMAND),CTRL.TYP) THEN
         	 				(*####################  DEBUG-MESSAGE  ###################################*)
          				(*IF _debug_enable THEN
            					LOG_CL.NEW_MSG := 'CE: #T:~1 #C:~2 #E:~3 #P:~6 #L:~7';
            					LOG_CL.PRINTF[1] := INT_TO_STRING(CTRL.TYP);
            					LOG_CL.PRINTF[2] := UINT_TO_STRING(CTRL.COUNT);
            					LOG_CL.PRINTF[3] := CTRL.ELEMENT;
            					LOG_CL.PRINTF[6] := CTRL.PATH;
            					LOG_CL.PRINTF[7] := UINT_TO_STRING(CTRL.LEVEL);
            					LOG_MSG();
          				END_IF;*)
          				(*########################################################################*)
					RETURN;
				ELSE
					EXIT;
				END_IF;
			END_IF;
			index := index + 1;
		END_WHILE;

	400: (* ---------- ATTRIBUTE SECTION ------------------ *)
		(* search first normal charakter *)
		WHILE (index <= stop AND BUF[index] <= BYTE#32) DO
			index := index + 1;
		END_WHILE;

		(* begin Attribe name *)
		e1 := 0;
		s1 := index;
		(* search end of Attrib Name '=' *)
		WHILE (index <= stop) DO
			IF BUF[index] = BYTE#61 THEN (* '=' Equals *)
				e1 := index - 1;
				EXIT;
			END_IF;
			index := index + 1;
		END_WHILE;

		IF e1 > 0 THEN
			(* Attribute Name *)
			CTRL.BLOCK1_START := INT_TO_UINT(s1);
			CTRL.BLOCK1_STOP  := INT_TO_UINT(e1);
			CTRL.ATTRIBUTE := OSCAT_BASIC.BUFFER_TO_STRING(PT:=ADR(BUF),SIZE:=INT_TO_UINT(STOP + 1),START:=CTRL.BLOCK1_START,STOP:=CTRL.BLOCK1_STOP);
			(* search end of Attrib Value '=' *)
			index := index + 2;
			e1 := 0;
			s1 := INDEX;
			WHILE (index <= stop AND e1 = 0) DO
				c := BUF[index];
				IF c = BYTE#34 OR c = BYTE#39 THEN (* " OR ' Equals *)
					e1 := index - 1;
				END_IF;
				index := index + 1;
			END_WHILE;

			IF e1 > 0 THEN
				(* Value *)
				CTRL.BLOCK2_START := INT_TO_UINT(s1);
				CTRL.BLOCK2_STOP  := INT_TO_UINT(e1);

				(* bei leeren "" ist start groesser als stop und wird somit zum leerstring *)
				CTRL.VALUE := OSCAT_BASIC.BUFFER_TO_STRING(PT:=ADR(BUF),SIZE:=INT_TO_UINT(stop + 1),START:=CTRL.BLOCK2_START,STOP:=CTRL.BLOCK2_STOP);
				(* search next non white space charakter *)
				WHILE (index <= stop AND BUF[index] <= BYTE#32) DO
					index := index + 1;
				END_WHILE;

					c := BUF[index];
					(* TagEnd '>' *)
					IF c = BYTE#62 THEN
						index := index + 1;
						index2 := index;

					(* search next non white space charakter *)
					WHILE (index <= stop AND BUF[index] <= BYTE#32) DO
						index := index + 1;
					END_WHILE;

					IF BUF[index] = BYTE#60 THEN (* TagBegin '<' *)
						mode := 100; (* -> NEXT-JOB: ELEMENT-SECTION *)
					ELSE
						index := index2;
						mode := 200; (* -> NEXT-JOB: TEXT-SECTION *)
					END_IF;

				ELSIF c = BYTE#47 OR c = BYTE#63 THEN (* TagTerm '/' OR '?' end Processing Instruction *)
					mode := 300; (* -> NEXT-JOB: END ELEMENT *)
				ELSE
					mode := 400; (* -> NEXT-JOB: ATTRIBUTE-SECTION *)
				END_IF;

				CTRL.COUNT := CTRL.COUNT + UINT#1;
				CTRL.TYP := 4;
				IF OSCAT_BASIC.BIT_OF_DWORD(WORD_TO_DWORD(command),CTRL.TYP) THEN
          				(*####################  DEBUG-MESSAGE  ###################################*)
          				(*IF _debug_enable THEN
            					LOG_CL.NEW_MSG := 'AT: #T:~1 #C:~2 #E:~3 #A:~4 #V:~5 #P:~6 #L:~7';
            					LOG_CL.PRINTF[1] := INT_TO_STRING(CTRL.TYP);
            					LOG_CL.PRINTF[2] := UINT_TO_STRING(CTRL.COUNT);
            					LOG_CL.PRINTF[3] := CTRL.ELEMENT;
            					LOG_CL.PRINTF[4] := CTRL.ATTRIBUTE;
            					LOG_CL.PRINTF[5] := CTRL.VALUE;
            					LOG_CL.PRINTF[6] := CTRL.PATH;
            					LOG_CL.PRINTF[7] := UINT_TO_STRING(CTRL.LEVEL);
            					LOG_MSG();
          				END_IF;*)
          				(*########################################################################*)
					RETURN;
				END_IF;
			END_IF;
		END_IF;

	500: (* ---------- SPECIAL DATA SECTION (Document Type Declarations) ---------- *)

		CTRL.TYP := 0;
		s1 := 0;
		index2 := 11;

		WHILE (s1 = 0) DO
			index2 := index2 + 1;
			CTRL.TYP := index2;

			CASE index2 OF
			12: (* CDATA *)
				s_code := '[CDATA[';
				e_code := ']]>';
			13: (* COMMENT *)
				s_code := '--';
				e_code := '-->';
			14: (* ANY DTD *)
				e_code := '';
				s1 := index;
				EXIT;
			END_CASE;

			e1 := LEN(s_code);
			IF OSCAT_BASIC.BUFFER_SEARCH(PT:=ADR(BUF),SIZE:=INT_TO_UINT(index + e1),STR:=S_CODE,POS:=index,IGN:=FALSE) = INDEX THEN
				s1 := index + e1;
			END_IF;
		END_WHILE;

		CTRL.BLOCK1_START := INT_TO_UINT(s1);
		IF LEN(e_code) > 0 THEN
			(* Ende Kennung suchen *)
			e1 := OSCAT_BASIC.BUFFER_SEARCH(PT:=ADR(BUF),SIZE:=INT_TO_UINT(stop + 1),STR:=e_code,POS:=index,IGN:=FALSE);
			CTRL.BLOCK1_STOP := INT_TO_UINT(e1 - 1);
			index := e1 + LEN(e_code); (* naechstes element *)
		ELSE
			(* suche '>' EndTag*)
			index2 := 1; (* <> Paar zähler *)
			WHILE (index <= stop AND index2 > 0) DO
				c := BUF[index];
				IF c = BYTE#60 THEN (* '<' TagBegin *)
					index2 := index2 + 1;
				ELSIF c = BYTE#62 THEN (* '>' TagEnd   *)
					index2 := index2 - 1;
				ELSIF c = BYTE#34 OR c = BYTE#39 THEN (* " Double Quote OR ' Single Quote *)
					index := index + 1;
					WHILE (index <= stop) DO
						c := BUF[index];
						IF c = BYTE#34 OR c = BYTE#39 THEN (* " Double Quote OR ' Single Quote *)
							EXIT;
						END_IF;
						index := index + 1;
					END_WHILE;
				END_IF;
				index := index + 1;
			END_WHILE;
			CTRL.BLOCK1_STOP := INT_TO_UINT(index - 2);
		END_IF;

		CTRL.VALUE := OSCAT_BASIC.BUFFER_TO_STRING(PT:=ADR(BUF),SIZE:=INT_TO_UINT(stop + 1),START:=CTRL.BLOCK1_START,STOP:=CTRL.BLOCK1_STOP);
		CTRL.COUNT := CTRL.COUNT + UINT#1;
		mode := 100; (* -> NEXT-JOB: ELEMENT *)

		IF OSCAT_BASIC.BIT_OF_DWORD(WORD_TO_DWORD(command),CTRL.TYP) THEN
      			(*####################  DEBUG-MESSAGE  ###################################*)
      			(*IF _debug_enable THEN
        				LOG_CL.NEW_MSG := 'DTD: #T:~1 #C:~2 #S:~3 #E:~4 #V:~5 #P:~6 #L:~7';
        				LOG_CL.PRINTF[1] := INT_TO_STRING(CTRL.TYP);
        				LOG_CL.PRINTF[2] := UINT_TO_STRING(CTRL.COUNT);
        				LOG_CL.PRINTF[3] := UINT_TO_STRING(CTRL.BLOCK1_START);
        				LOG_CL.PRINTF[4] := UINT_TO_STRING(CTRL.BLOCK1_STOP);
        				LOG_CL.PRINTF[5] := CTRL.VALUE;
        				LOG_CL.PRINTF[6] := CTRL.PATH;
        				LOG_CL.PRINTF[7] := UINT_TO_STRING(CTRL.LEVEL);
        				LOG_MSG();
      			END_IF;*)
      			(*########################################################################*)
			RETURN;
		END_IF;

	END_CASE;
END_WHILE;


(* revision history
ks	18. oct. 2008	rev 1.0
	original version

ks	20. oct. 2009	rev 1.1
	Networkbuffer und Buffer-funktionen auf Basis 0

ks	10. mai. 2010	rev 1.2
	stringlänge maximal 250 zeichen

*)

END_FUNCTION_BLOCK

// POUs/NETWORK/DNS_REV_CLIENT
FUNCTION_BLOCK DNS_REV_CLIENT
VAR_IN_OUT
	IP_C : IP_C; (* IP_Control Verwaltungsstruktur *)
	S_BUF : NETWORK_BUFFER;
	R_BUF : NETWORK_BUFFER;
END_VAR
VAR_INPUT
	ACTIVATE : BOOL;
	IP4 : DWORD;
	IP4_DNS : DWORD;
END_VAR
VAR_OUTPUT
	DOMAIN : STRING;
	DONE : BOOL;
	ERROR : DWORD;
END_VAR
VAR
	IP_FIFO : IP_FIFO;
	ip_state : BYTE;
	ip_id : BYTE;
	state : INT;
	ip4_copy : DWORD;
	d : STRING(27);
	activate_last : BOOL;
	i : INT;
	dl : INT;
	p1 : INT;
	char : BYTE;
	char_count : INT;
	tid : BYTE;
END_VAR

(*
version 1.0	28. dec. 2009
programmer 	ks
tested BY	ks

DNS_REV_CLIENT führt eine Reverse-Domain-Name Abfrage durch, und ermittelt aus einer IP-Adresse den zugehörigen Domain-Namen.

*)

(* Domain Name System (query) *)

CASE state OF
00: (* auf positive Flanke GET warten *)
	IF ACTIVATE AND NOT activate_last THEN
		ERROR := DWORD#0;
		ip4_copy := ip4; (* IP4 sichern *)
		ip_state := BYTE#1;
		DOMAIN := '';
		DONE := FALSE;

		d := '';
		FOR i := 1 TO 4 DO
			d := CONCAT(d,BYTE_TO_STRING(DWORD_TO_BYTE(IP4)));
			d := CONCAT(d,'.');
			IP4 := ROR(IP4,8);
		END_FOR;
		d := CONCAT(d,'in-addr.arpa');
		state := 10;
	END_IF;

10: (* Bei IP_Control anmelden *)
	IF ip_state = BYTE#3 THEN
		dl := LEN(d);

		(* sendebuffer initialisieren *)
		char_count := 17 + dl;
		FOR i := 0 TO char_count DO
			S_BUF.BUFFER[i] := BYTE#00;
		END_FOR;

		tid := UINT_TO_BYTE(BYTE_TO_UINT(tid) + UINT#1);
		S_BUF.BUFFER[01] := tid; (* Transaction ID lowbyte *)
		S_BUF.BUFFER[02] := BYTE#16#01; (* Flags: highbyte *)
		S_BUF.BUFFER[05] := BYTE#16#01; (* Questions: lowbyte *)

		(* den servernamen von hinten nach vorne bearbeiten *)
		i := dl + 12;
		char_count := 0;

		WHILE i > 12 DO
			char := OSCAT_BASIC.CODE(STR:=d,POS:=i - 12);

			(* prüfe auf haupt/sub domänen namens-teiler "." *)
			IF char = BYTE#46 THEN
				(* anstelle des teilers "." wird die länge des erkannten haupt/sub domänennames eingetragen *)
				S_BUF.BUFFER[i] := INT_TO_BYTE(char_count);
				char_count := 0;
			ELSE
				S_BUF.BUFFER[i] := char; (* char in buffer eintragen *)
				char_count := char_count + 1; (* anzahl char zählen *)
			END_IF;
			i := i - 1;
		END_WHILE;

		S_BUF.BUFFER[i] := INT_TO_BYTE(char_count); (* längenangabe des ganz linken (ersten) domänennamens eintragen *)
		i := dl + 15; (* position hinter dem servernamen *)
		S_BUF.BUFFER[i] := BYTE#12; (* Type: PTR (Domain name pointer) lowbyte *)
		i := i + 2;
		S_BUF.BUFFER[i] := BYTE#01; (* Class: IN lowbyte *)
		i := i + 1;

		(* IP Datenverkehr einrichten *)
		IP_C.C_PORT := WORD#53; (* Portnummer eintragen *)
		IP_C.C_IP := IP4_DNS; (* IP eintragen *)
		IP_C.C_MODE := BYTE#1; (* Mode: UDP+AKTIV+PORT+IP *)
		IP_C.C_ENABLE := TRUE; (* Verbindungsaufbau freigeben *)
		IP_C.TIME_RESET := TRUE; (* Zeitueberwachung rücksetzen *)
		IP_C.R_OBSERVE  := TRUE; (* Datenempfang ueberwachen *)
		S_BUF.SIZE := INT_TO_UINT(i); (* sendelänge eintragen *)
		R_BUF.SIZE := UINT#0; (* Empfangslänge rücksetzen *)
		state := 30;
	END_IF;

30:
	IF IP_C.ERROR <> DWORD#00 THEN
		ERROR := IP_C.ERROR;
	(* prüfe ob antwort telegramm die richtige Transaction-ID und mindestlänge hat *)
	ELSIF (S_BUF.SIZE = UINT#0) AND (tid = R_BUF.BUFFER[1]) AND (R_BUF.SIZE >= INT_TO_UINT(i+12)) THEN

		(* prüfe Return code der Flags. 4 bits *)
		ERROR := BYTE_TO_DWORD(R_BUF.BUFFER[3] AND BYTE#2#0000_1111);

		IF ERROR = DWORD#00 THEN

			i := R_BUF.SIZE - 2;
			WHILE R_BUF.BUFFER[i] > 0 DO
				IF i = 0 THEN EXIT; END_IF;
				i := i - 1;
			END_WHILE;

			i := i + 2;
			p1 := i + 1;
			WHILE i < R_BUF.SIZE DO
				dl := R_BUF.BUFFER[i];
				IF dl > 0 THEN
					R_BUF.BUFFER[i] := BYTE#46;
					i := i + dl + 1;
				ELSE
					DOMAIN := OSCAT_BASIC.BUFFER_TO_STRING(PT:=ADR(R_BUF.BUFFER),SIZE:=SIZEOF(R_BUF.BUFFER),START:=p1,STOP:=i-1);
					EXIT;
				END_IF;
			END_WHILE;
			state := 0;
			DONE := TRUE;
		END_IF;
	END_IF;

	IF ERROR <> DWORD#0 THEN
		state := 0;
	END_IF;

	IF state = 0 THEN
		IP_C.R_OBSERVE := FALSE; (* Datenempfang ueberwachen *)
		ip_state := BYTE#4; (* Abmelden *)
	END_IF;

END_CASE;

activate_last := ACTIVATE; (* letzten Status sichern zur Flankenerkennung *)

(* IP_FIFO *)
IP_FIFO(FIFO:=IP_C.FIFO,STATE:=ip_state,ID:=ip_id);

(* revision history

ks	28. dec. 2009	rev 1.0
	original version

*)


(*----------------------------------------------------------------------------------------------------------------*)
(* Flags: 0x0100 (Standard query)                                                                                            *)
(* 0... .... .... .... = Response: Message is a query                                                                   *)
(* .000 0... ....  = Opcode: Standard query (0)                                                                          *)
(* .... ..0. .... .... = Truncated: Message is not truncated                                                          *)
(* .... ...1 .... .... = Recursion desired: Do query recursively                                                    *)
(* .... .... .0.. .... = Z: reserved (0)                                                                                                  *)
(* .... .... ...0 .... = Non-authenticated data OK: Non-authenticated data is unacceptable *)
(*-----------------------------------------------------------------------------------------------------------------*)

(*
Errorcodes  Description	References 
000	No error. 		 	The request completed successfully.
001	Format error. 		The name server was unable to interpret the query. 
002	Server failure.  	The name server was unable to process this query due to a problem with the name server. 
003	Name Error. 	 	Meaningful only for responses from an authoritative name server, this code signifies that the domain name referenced in the query does not exist.
004	Not Implemented. 	The name server does not support the requested kind of query.
005	Refused. 			The name server refuses to perform the specified operation for policy reasons.
  						 For example, a name server may not wish to provide the information to the particular requester, or a name server may not wish to perform a particular operation (e.g., zone transfer) for particular data.
006	YXDomain.			Name Exists when it should not. 
007	YXRRSet. RR			Set Exists when it should not. 
008	NXRRSet. RR			Set that should exist does not. 
009	NotAuth.			Server Not Authoritative for zone. 
010	NotZone,			Name not contained in zone. 
255	Timeout				No Response  
*)

END_FUNCTION_BLOCK

// POUs/NETWORK/GET_WAN_IP
FUNCTION_BLOCK GET_WAN_IP
VAR_IN_OUT
	IP_C : IP_C; (* IP_Control Verwaltungsstruktur *)
	S_BUF : NETWORK_BUFFER;
	R_BUF : NETWORK_BUFFER;
END_VAR
VAR_INPUT
	ACTIVATE : BOOL;
END_VAR
VAR_OUTPUT
	WAN_IP4 : DWORD;
	DONE : BOOL;
	NEW_IP4 : BOOL;
	ERROR_C : DWORD;
	ERROR_T : BYTE;
END_VAR
VAR
	URL_DATA : url;
	DNS_CLIENT : DNS_CLIENT;
	HTTP_GET : HTTP_GET;
	activate_last : BOOL;
	wan_ip4_last : DWORD;
	state : INT;
	st_ip : STRING(120);
	i1 :	INT;
	p1 : INT;
	p2 : INT;
	p3 : INT;
END_VAR

(*
version 1.1	28. dec. 2009
programmer 	ks
tested by	ks

GET_WAN_IP ermittelt die aktuelle WAN-IP (Internet-Adresse)
*)

CASE state OF

00:
	IF ACTIVATE AND NOT activate_last THEN
		state := 20;
		DONE := FALSE;
		ERROR_C := DWORD#0;
		ERROR_T := BYTE#0;
	END_IF;

20: (* URL for DNS UND HTTP-GET *)
	URL_DATA := STRING_TO_URL(STR:='checkip.dyndns.com',DEFAULT_PROTOCOL:='',DEFAULT_PATH:='');
	state := 40;

40:
	IF DNS_CLIENT.DONE THEN
		state := 60;
	ELSIF (DNS_CLIENT.ERROR > DWORD#00) THEN
		(* Fehlerbehandlung *)
		ERROR_C := DNS_CLIENT.ERROR;
		ERROR_T := BYTE#01;
		state := 100;
	END_IF;

60:
	IF HTTP_GET.DONE THEN
		state := 80;
	ELSIF (HTTP_GET.ERROR > DWORD#00) THEN
		(* Fehlerbehandlung *)
		ERROR_C := HTTP_GET.ERROR;
		ERROR_T := BYTE#02;
		state := 100;
	END_IF;

80:
	(* Als Antwort wird folgende HTML Seite empfangen , hier muss die IP-Adresse herauskopiert werden *)
	(* <html><head><title>Current IP Check</title></head><body>Current IP Address: 85.127.217.33</body></html> *)
	st_ip := '';
	p1 := 0;
	FOR i1 := UINT_TO_INT(HTTP_GET.BODY_START) TO UINT_TO_INT(HTTP_GET.BODY_STOP) DO
		IF R_BUF.BUFFER[i1] = BYTE#58 THEN (* suche ':' *)
			p1 := i1 + 2;
			EXIT;
		END_IF;
	END_FOR;

	p3 := p1 + 15;
	IF p1 > 0 AND p3 < UINT_TO_INT(HTTP_GET.BODY_STOP) THEN
		FOR p2 := p1 TO p3 DO
			IF R_BUF.BUFFER[p2] <> BYTE#60 THEN (* suche '<' *)
				st_ip := CONCAT(st_ip,OSCAT_BASIC.CHR_TO_STRING(C:=R_BUF.BUFFER[p2]));
			ELSE
				EXIT;
			END_IF;
		END_FOR;
	END_IF;

	WAN_IP4 := IP4_DECODE(STR:=st_ip);

	IF WAN_IP4 <> DWORD#0 THEN
		DONE := TRUE;
		NEW_IP4 := WAN_IP4 <> wan_ip4_last;
		wan_ip4_last := WAN_IP4;
	ELSE
		ERROR_C := DWORD#01; (* keine gültige IP gefunden *)
		ERROR_T := BYTE#03;
	END_IF;
	state := 100;

100:
	(* UNLOCK HTTP DATA *)
	IF (NOT HTTP_GET.DONE) THEN
		state := 0;
		DONE := ERROR_T = BYTE#0;
	END_IF;

END_CASE;

(* ---------------- DNS --------------- *)
DNS_CLIENT(	IP_C:=IP_C,
			S_BUF:=S_BUF,
			R_BUF:=R_BUF,
			DOMAIN:=URL_DATA.DOMAIN,
			IP4_DNS:=DWORD#00,
			ACTIVATE:=state=40 (* DNS Start *)
			);
(* nicht oder nicht direkt verwendete Parameter *)
(* DWORD :=DNS_CLIENT.IP4;
   BOOL  :=DNS_CLIENT.DONE;
   BYTE  :=DNS_CLIENT.ERROR; *)
(* -------------------------------------*)

(* ------------- HTTP_GET --------------- *)

HTTP_GET(	IP_C:=IP_C,
			S_BUF:=S_BUF,
			R_BUF:=R_BUF,
			IP4:=DNS_CLIENT.IP4,
			GET:=state=60,
			MODE:=BYTE#2, (* HTTP 1.1 mit persistenter Verbindung *)
			UNLOCK_BUF:=state=100,
			URL_DATA:=URL_DATA
			);

(* nicht oder nicht direkt verwendete Parameter *)
(*STRING := HTTP_GET.HTTP_STATUS;
  UINT :=HTTP_GET.HEADER_START;
  UINT :=HTTP_GET.HEADER_STOP;
  UINT :=HTTP_GET.BODY_START;
  UINT :=HTTP_GET.BODY_STOP;
  BOOL :=HTTP_GET.DONE;
  BYTE :=HTTP_GET.ERROR;
*)
(* -------------------------------------*)

activate_last := ACTIVATE;

(* revision history
ks	28. dec 2009	rev 1.1
	original version

*)

END_FUNCTION_BLOCK

// POUs/CONVERT/HTML_DECODE
FUNCTION HTML_DECODE : STRING(OSCAT_BASIC.STRING_LENGTH)
VAR_INPUT
	IN : STRING(OSCAT_BASIC.STRING_LENGTH);
END_VAR
VAR
	pos : INT;
	end : INT;
	tmp : STRING(10);
	code : STRING(1);
END_VAR

(*
version 1.3		10. may 2010
programmer 	hugo
tested by		oscat

HTML_DECODE converts HTML coded characters to text. 
&amp; is replaced by & ("Ampersand")
&lt; is replaced by < ("lower than")
&gt; is replaced by > ("greater than")
&quot; is replaced by " ("Quote")
all other &names characters are replaced by their respective character codes.

*)

HTML_DECODE := IN;

(* docode characters encoded by character position *)
pos := FIND(HTML_DECODE, '&');
WHILE pos > 0 DO
	tmp := MID(HTML_DECODE, 2, pos + 1);
	IF tmp = '#x' OR tmp = '#X' THEN
		(* hexadecimal representation found *)
		tmp := MID(HTML_DECODE, 10, pos + 3);
		end := FIND(tmp, ';');
		CODE := OSCAT_BASIC.CHR_TO_STRING(DWORD_TO_BYTE(OSCAT_BASIC.HEX_TO_DWORD(LEFT(tmp, end - 1))));
		HTML_DECODE := REPLACE(HTML_DECODE, CODE, end + 3, pos);
	ELSIF LEFT(tmp,1) = '#' THEN
		tmp := MID(HTML_DECODE, 10, pos + 2);
		end := FIND(tmp, ';');
		CODE := OSCAT_BASIC.CHR_TO_STRING(INT_TO_BYTE(STRING_TO_INT(LEFT(tmp, end - 1))));
		HTML_DECODE := REPLACE(HTML_DECODE, CODE, end + 2, pos);
	ELSE
		(* replace all named characters *)
		tmp := MID(HTML_DECODE, 10, pos + 1);
		end := FIND(tmp, ';');
		CODE := OSCAT_BASIC.CHR_TO_STRING(OSCAT_BASIC.CHARCODE(LEFT(tmp, end - 1)));
		HTML_DECODE := REPLACE(HTML_DECODE, CODE, end + 1, pos);
	END_IF;
	(* search for next occurence of encoded characters *)
	pos := OSCAT_BASIC.FINDP(HTML_DECODE, '&', pos + 1);
END_WHILE;



(* revision history
hm	3. mai. 2008	rev 1.0
	original version

hm	16. jun. 2008	rev 1.1
	changed nested call of replace for better compatibility

hm	17. dec. 2008	rev 1.2
	changed function CHR to CHR_TO_STRING

hm	10. may. 2010	rev 1.3
	stringlength 250

*)

END_FUNCTION

// POUs/CONVERT/HTML_ENCODE
FUNCTION HTML_ENCODE : STRING(OSCAT_BASIC.STRING_LENGTH)
VAR_INPUT
	IN : STRING(OSCAT_BASIC.STRING_LENGTH);
	M : BOOL;
END_VAR
VAR
	pt_in : POINTER TO ARRAY[1..255] OF BYTE;
	pt_out : POINTER TO ARRAY[1..256] OF BYTE;
	pos_in : INT;
	pos_out : INT;
	stop : INT;
	B: BYTE;
	tmp : STRING(10);
	i: INT;
END_VAR


(*
version 1.1		10. may. 2010
programmer 	hugo
tested by		hugo 

HTML_ENCODE checks a string if it contains reserved HTML characters and converts them to alternative html coding.
& is replaced by &amp; ("Ampersand")
< is replaced by &lt; ("lower than")
> is replaced by &gt; ("greater than")
" is replaced by &quot; ("Quote")

*)

pt_in  := ADR(in);
pt_out := ADR(HTML_ENCODE);

(* scan the input string and convert unallowed characters *)
pos_in := 1;
stop := LEN(in);
FOR pos_out := 1 TO 250 DO
	IF pos_in > stop THEN EXIT; END_IF;
	B := pt_in^[pos_in];
	CASE BYTE_TO_INT(B) OF
		34: (* " detected *)
			IF pos_out > OSCAT_BASIC.STRING_LENGTH - 6 THEN EXIT; END_IF;
			pt_out^[pos_out] := 38;
			pos_out := pos_out + 1;
			pt_out^[pos_out] := 113;
			pos_out := pos_out + 1;
			pt_out^[pos_out] := 117;
			pos_out := pos_out + 1;
			pt_out^[pos_out] := 111;
			pos_out := pos_out + 1;
			pt_out^[pos_out] := 116;
			pos_out := pos_out + 1;
			pt_out^[pos_out] := 59;
		38: (* & detected *)
			IF pos_out > OSCAT_BASIC.STRING_LENGTH - 5 THEN EXIT; END_IF;
			pt_out^[pos_out] := 38;
			pos_out := pos_out + 1;
			pt_out^[pos_out] := 97;
			pos_out := pos_out + 1;
			pt_out^[pos_out] := 109;
			pos_out := pos_out + 1;
			pt_out^[pos_out] := 112;
			pos_out := pos_out + 1;
			pt_out^[pos_out] := 59;
		60: (* < detected *)
			IF pos_out > OSCAT_BASIC.STRING_LENGTH - 4 THEN EXIT; END_IF;
			pt_out^[pos_out] := 38;
			pos_out := pos_out + 1;
			pt_out^[pos_out] := 108;
			pos_out := pos_out + 1;
			pt_out^[pos_out] := 116;
			pos_out := pos_out + 1;
			pt_out^[pos_out] := 59;
		62: (* > detected *)
			IF pos_out > OSCAT_BASIC.STRING_LENGTH - 4 THEN EXIT; END_IF;
			pt_out^[pos_out] := 38;
			pos_out := pos_out + 1;
			pt_out^[pos_out] := 103;
			pos_out := pos_out + 1;
			pt_out^[pos_out] := 116;
			pos_out := pos_out + 1;
			pt_out^[pos_out] := 59;
	ELSE
		IF M AND B > 127 THEN
			tmp :=OSCAT_BASIC. CHARNAME(B);
			(* exit if output string has not enough space *)
			IF pos_out + LEN(tmp) + 2 <= 250 THEN
				pt_out^[pos_out] := 38;
				pos_out := pos_out + 1;
				FOR i := 1 TO LEN(tmp) DO
					pt_out^[pos_out] := OSCAT_BASIC.CODE(tmp, i);
					pos_out := pos_out + 1;
				END_FOR;
				pt_out^[pos_out] := 59;
			END_IF;
		ELSE
			pt_out^[pos_out] := B;
		END_IF;
	END_CASE;
	(* increment in by 1 *)
	pos_in := pos_in + 1;
END_FOR;

(* terminate the output string *)
pt_out^[pos_out] := 0;



(* revision history
hm		3. mai. 2008	rev 1.0
	original version

hm		10. mai. 2008	rev 1.1
	stringlength 250
*)

END_FUNCTION

// POUs/NETWORK/IP2GEO
FUNCTION_BLOCK IP2GEO
VAR_IN_OUT
	IP_C : IP_C; (* IP_Control Verwaltungsstruktur *)
	S_BUF : NETWORK_BUFFER;
	R_BUF : NETWORK_BUFFER;
	GEO : IP2GEO_DATA;
END_VAR
VAR_INPUT
	IP : DWORD;
	ACTIVATE : BOOL;
END_VAR
VAR_OUTPUT
	BUSY : BOOL;
	DONE : BOOL;
	ERROR_C : DWORD;
	ERROR_T : BYTE;
END_VAR
VAR
	CTRL : XML_CONTROL;
	XML_READER : XML_READER;
	URL_DATA : url;
	DNS_CLIENT : DNS_CLIENT;
	HTTP_GET : HTTP_GET;
	last_state : BOOL;
	value_int :	INT;
	value_real : REAL;
	v_real : REAL;
	state : INT;
END_VAR
(*

version 	1.1	07.oct. 2010
programmer 	ks
tested by	ks

IP2GEO ermittelt die aktuelle WAN-IP und die dazugehörigen geographischen Infos

zusatzinfos: http://www.worldtimezone.com/time/wtzresult.php?CiID=10182&forma=

example:

http://ipinfodb.com/ip_query.php?timezone=true&IP=

<?xml version="1.0" encoding="UTF-8" ?> 
- <Response>
  <Ip>85.127.218.109</Ip> 
  <Status>OK</Status> 
  <CountryCode>AT</CountryCode> 
  <CountryName>Austria</CountryName> 
  <RegionCode>09</RegionCode> 
  <RegionName>Wien</RegionName> 
  <City>Vienna</City> 
  <ZipPostalCode /> 
  <Latitude>48.2</Latitude> 
  <Longitude>16.3667</Longitude> 
  <TimezoneName>Europe/Vienna</TimezoneName> 
  <Gmtoffset>7200</Gmtoffset> 
  <Isdst>1</Isdst> 
  </Response>

*)

CASE state OF

00:
	IF ACTIVATE AND NOT last_state THEN
		state := 20;
		DONE := FALSE;
		BUSY := TRUE;
		ERROR_C := DWORD#0;
		ERROR_T := BYTE#0;
	END_IF;

20: (* URL for DNS UND HTTP-GET *)
	(* Example: http://ipinfodb.com/ip_query.php?ip=10.10.10.10 *)
	(* Example: http://ipinfodb.com/ip_query.php?timezone=true&IP=*)
	URL_DATA:=STRING_TO_URL(STR:='http://ipinfodb.com/ip_query.php?timezone=true&IP=',DEFAULT_PROTOCOL:='',DEFAULT_PATH:='');

	IF IP > DWORD#0 THEN
		URL_DATA.QUERY := CONCAT(URL_DATA.QUERY,IP4_TO_STRING(IP4:=IP));
	END_IF;

	state := 40;

40:
	IF DNS_CLIENT.DONE THEN
		state := 60;
	ELSIF (DNS_CLIENT.ERROR > DWORD#00) THEN
		(* Fehlerbehandlung *)
		ERROR_C := DNS_CLIENT.ERROR;
		ERROR_T := BYTE#01;
		state := 100;
	END_IF;

60:
	IF HTTP_GET.DONE THEN
		state := 80;
		CTRL.START_POS := HTTP_GET.BODY_START;
		CTRL.STOP_POS := HTTP_GET.BODY_STOP;
		CTRL.COMMAND := WORD#2#10000000_00011000; (* ONLY TEXT AND ATTRIBUTE *)
		CTRL.WATCHDOG := T#1ms;

	ELSIF (HTTP_GET.ERROR > DWORD#00) THEN
		(* Fehlerbehandlung *)
		ERROR_C := HTTP_GET.ERROR;
		ERROR_T := BYTE#02;
		state := 100;
	END_IF;

80:
	(* XML Daten seriell lesen *)
	XML_READER(CTRL:=CTRL,BUF:=R_BUF.BUFFER);
	IF CTRL.TYP < 98 THEN (* nur auswerten wenn kein Watchdog durchlauf *)
		(* automatische konvertierung in real und int ausführen *)
		value_int := 0;
		value_real := 0.0;
		IF LEN(CTRL.VALUE) <= 20 THEN
			v_real :=OSCAT_BASIC.FLOAT_TO_REAL(FLT:=CTRL.VALUE);
			IF OSCAT_BASIC.CHK_REAL(v_real) = 0 THEN (* !!! prüft auf gültigen REAL Wert, ansonsten stürzt Twincat ab !!!!  *)
				value_real := v_real;
				value_int := REAL_TO_INT(value_real);
			END_IF;
		END_IF;

		CASE UINT_TO_INT(CTRL.COUNT) OF

		07: GEO.IP4 := IP4_DECODE(STR:=CTRL.VALUE); (* IP-Adresse *)
		10: GEO.STATE := 'OK' = CTRL.VALUE; (* STATUS *)
		13: GEO.COUNTRY_CODE := CTRL.VALUE; (* Country-Code *)
		16: GEO.COUNTRY_NAME := CTRL.VALUE; (* Country-Name *)
		19: GEO.REGION_CODE := CTRL.VALUE; (* Region-Code *)
		22: GEO.REGION_NAME := CTRL.VALUE; (* Region-Name *)
		25: GEO.CITY := CTRL.VALUE; (* City *)
		31: GEO.GEO_LATITUDE := value_real; (* Latitude *)
		34: GEO.GEO_LONGITUDE := value_real; (* Longitude *)
		37: GEO.TIME_ZONE_NAME := CTRL.VALUE; (* TimeZone Name *)
		40: GEO.GMT_OFFSET := value_int; (* GMT OFFSET in Sekunden *)
		43: GEO.IS_DST := value_int > 0; (* Sommerzeit aktiv *)
		END_CASE;

	ELSIF CTRL.TYP = 99 THEN (* EXIT - letztes Element gelesen *)
		DONE := TRUE;
		state := 100;
	END_IF;

100:
	(* UNLOCK HTTP DATA *)
	IF (NOT HTTP_GET.DONE) THEN
		state := 0;
		BUSY := FALSE;
		DONE := ERROR_T = BYTE#0;
	END_IF;

END_CASE;

(* ---------------- DNS --------------- *)
DNS_CLIENT(	IP_C:=IP_C,
			S_BUF:=S_BUF,
			R_BUF:=R_BUF,
			DOMAIN:=URL_DATA.DOMAIN,
			IP4_DNS:=DWORD#00,
			ACTIVATE:=state=40 (* DNS Start *)
			);

(* nicht oder nicht direkt verwendete Parameter *)
(* 	DWORD :=DNS_CLIENT.IP4;
	BOOL  :=DNS_CLIENT.DONE;
	BYTE  :=DNS_CLIENT.ERROR; *)
(* -------------------------------------*)

(* ------------- HTTP_GET --------------- *)
HTTP_GET(	IP_C:=IP_C,
			S_BUF:=S_BUF,
			R_BUF:=R_BUF,
			IP4:=DNS_CLIENT.IP4,
			GET:=state=60,
			MODE:=BYTE#2, (* HTTP 1.1 mit persistenter Verbindung *)
			UNLOCK_BUF:=state=100,
			URL_DATA:=URL_DATA
			);

(* nicht oder nicht direkt verwendete Parameter *)
(*	STRING := HTTP_GET.HTTP_STATUS;
	UINT :=HTTP_GET.HEADER_START;
	UINT :=HTTP_GET.HEADER_STOP;
	UINT :=HTTP_GET.BODY_START;
	UINT :=HTTP_GET.BODY_STOP;
	BOOL :=HTTP_GET.DONE;
	BYTE :=HTTP_GET.ERROR;
*)
(* -------------------------------------*)

last_state := ACTIVATE;

(* revision history
ks	14. aug. 2009	rev 1.0
	original version

ks	07. oct. 2010	rev 1.1
	new url , ip2geo fields , REAL_CHECK
*)

END_FUNCTION_BLOCK

// POUs/CONVERT/IP4_CHECK
FUNCTION IP4_CHECK : BOOL
VAR_INPUT
	NIP : DWORD;
	LIP : DWORD;
	SM : DWORD;
END_VAR


(*
version 1.0	4. mar 2008
programmer 	hugo
tested by		oscat

IP4_CHECK testet ob eine Network IP und Local_IP im selben Subnet sind.

*)

IP4_CHECK := (NIP AND sm) = (LIP AND SM);


(* revision history
hm		4. mar 2008	rev 1.0
	original version

*)

END_FUNCTION

// POUs/HARDWARE/IP_CONTROL2_V2
FUNCTION_BLOCK IP_CONTROL2_V2
VAR_IN_OUT
	IP_C : IP_C; (* IP_Control Verwaltungsstruktur *)
	S_BUF : NETWORK_BUFFER_SHORT; (* Externer Sendbuffer *)
	R_BUF : NETWORK_BUFFER_SHORT; (* Externer Receivebuffer *)
END_VAR
VAR_INPUT
	IP : DWORD; (* IP Adresse *)
	PORT : WORD; (* Port Nummer *)
	TIME_OUT : TIME; (* Ueberwachungszeit Connect / Send / Receive *)
END_VAR
VAR
	c_time : UDINT; (* CONNECT-Time (Zeit bei nicht vorhandener Verbindung) *)
	s_time : UDINT; (* SEND-Time    (Zeit seit letzten Datensenden) *)
	r_time : UDINT; (* RECEIVE-Time (Zeit seit letztem Datenempfang) *)

	c_enable : BOOL; (* Connect: freigabe *)
	c_ip : DWORD; (* Connect: aktuelle IP-Adresse *)
	c_port : WORD; (* Connect: aktuelle Port-Nummer *)
	c_mode : BYTE; (* Connect: aktueller Mode UDP/TCP...... *)
	c_status : BYTE; (* Connect: Status (Errorcode) *)
	c_ready : BOOL; (* Connect: Verbindung aufgebaut *)
	c_ready_old : BOOL; (* Connect: letzter Zustand von c_ready für Flankenauswertung *)
	c_select : BOOL; (* non blocking mode - abfrage über select durchführen *)
	c_fdWrite : SOCKET_FD_SET;
	c_Timeout : SOCKET_TIMEVAL;

	s_total : INT; (* Send: Gesamtanzahl Bytes zum senden *)
	s_cur_pos : INT; (* Send: aktuelle Sendeposition *)
	s_cur_size : INT; (* Send: aktuelle Sendegroesse *)
	s_max_size : INT; (* Send: maximale Telegrammlänge fuer Senden *)
	s_start : BOOL; (* Send: Sende modus aktivieren *)
	s_active : BOOL; (* Send: Daten senden ist aktiv *)
	s_req : BOOL; (* Send: Start Daten senden *)
	s_done : BOOL; (* Send: ohne Fehler beendet *)
	s_status : BYTE; (* Send: Status (Errorcodes) *)

	r_status : BYTE; (* Receive: Status (Errorcodes) *)
	r_count : INT; (* Receive: Anzahl empfangener Bytes *)
	r_offset : INT; (* Receive: aktuelle Position in externen Receivebuffer *)
	r_max_size : INT; (* Receive: groesse des externen Empfangbuffers*)

	new_connection : BOOL; (* Neue Verbindungsparameter vorhanden *)
	tx : DWORD; (* letzter zeitwert *)
	error_time : DWORD; (* aktueller Timeout-Wert *)

	state: BYTE; (* schrittmerker für connect *)
	server_socket :  RTS_IEC_HANDLE:= RTS_INVALID_HANDLE;
	socket : RTS_IEC_HANDLE:= RTS_INVALID_HANDLE;
	sockaddr : SOCKADDRESS;
	sockaddr_size : DWORD;
	plc_841 : BOOL;
	plc_881 : BOOL;
	dint_true : DINT := 1;
	bytes_received : DINT;
	bytes_sent : DINT;
	udp_mode : BOOL;

	(*LOG_MSG : LOG_MSG;
	_debug_enable : BOOL := TRUE;
	debug_index : INT;
	debug_ID : INT;
	debug_lasterror : DWORD;
	debug_last_id : INT := 255;
	state_last: BYTE;*)

END_VAR

VAR CONSTANT
	STOP : BYTE := 0;
	TS_INIT: BYTE := 1;
	TS_OPEN : BYTE:= 2;
	UDP_INIT : BYTE:= 31;
	TC_INIT : BYTE:= 51;
	TC_CONNECT : BYTE:= 52;
	C_WAIT : BYTE:= 250;
	C_CLOSE : BYTE:= 251;
END_VAR

(*

version 1.9		26. Feb. 2012
programmer 		ks
tested by			ks

IP_CONTROL ist ein Wrapper-Baustein um eine Hersteller neutrale Schnittstelle zum Ethernet zu schaffen
*)

(* ---------------------- Debug-Message ----------------------------*)
(*IF _debug_enable THEN
	IF IP_C.FIFO.ID > BYTE#0 THEN
		debug_index := IP_C.FIFO.NR;
		debug_ID := BYTE_TO_INT(IP_C.FIFO.X[debug_index]);
	END_IF;
END_IF;*)
(* -----------------------------------------------------------------------------*)

(* read system time *)
tx := OSCAT_BASIC.T_PLC_MS();

IF IP_C.C_PORT = 0 THEN
	IP_C.C_PORT := PORT; (* uebergebenen PORT durch parametrierten PORT ersetzen *)
END_IF;
IF IP_C.C_IP = 0 AND IP_C.C_MODE < 4 THEN
	IP_C.C_IP := IP; (* uebergebene IP durch paramtrierte IP ersetzen *)
END_IF;

new_connection := c_ip <> IP_C.C_IP OR c_mode <> IP_C.C_MODE OR c_port <> IP_C.C_PORT; (* neue Verbindungs erwünscht ? *)
c_enable := IP_C.C_ENABLE AND NOT new_connection;

IF IP_C.C_ENABLE AND IP_C.ERROR = 0 AND state = STOP THEN (* Freigabe,kein Fehler,kein Socket offen *)
	c_ip   := IP_C.C_IP;
	c_mode := IP_C.C_MODE;
	c_port := IP_C.C_PORT;
	plc_841 := ADR(%MW0)=16#30000000; (*750-841*)
	plc_881 := ADR(%MW0)=16#20000000; (*750-881*)
	udp_mode := C_MODE.0; (* Mode 1,3,5 = udp *)

	error_time := TIME_TO_DWORD(MAX(T#200ms,TIME_OUT));
	IP_C.TIME_RESET := TRUE; (* Alle Timer ruecksetzen *)

	r_max_size := SIZEOF(R_BUF.BUFFER);
	s_max_size := SIZEOF(S_BUF.BUFFER);

	IF C_MODE.0 THEN (* Mode: 1,3,5 = UDP CLIENT/SERVER *)
		state := UDP_INIT;
	ELSIF C_MODE = 0 THEN (* Mode: 0 = TCP CLIENT *)
		state := TC_INIT;
	ELSE
		state := TS_INIT; (* Mode: 2,4 = TCP SERVER *)
	END_IF;

	(* ---------------------- Debug-Message ----------------------------*)
	(*IF _debug_enable THEN
		LOG_CL.NEW_MSG := 'IP_CON: MODE ~1 / IP ~2 / PORT ~3 /ID ~6';
		LOG_CL.PRINTF[1] := BYTE_TO_STRING(C_MODE);
		LOG_CL.PRINTF[2] := IP4_TO_STRING(c_ip);
		LOG_CL.PRINTF[3] := WORD_TO_STRING(c_port);
		LOG_CL.PRINTF[6] := INT_TO_STRING(debug_ID);
		LOG_MSG();
	END_IF;*)
	(* -----------------------------------------------------------------------------*)

END_IF;

(* ---------------------- Debug-Message ----------------------------*)
(*IF  _debug_enable THEN
	IF state <> state_last THEN
		LOG_CL.NEW_MSG := 'IP_STEP ~1 -IP_ID ~6';
		LOG_CL.PRINTF[1] := BYTE_TO_STRING(state);
		LOG_CL.PRINTF[6] := INT_TO_STRING(debug_ID);
		LOG_MSG();
		state_last := state;
	END_IF;
END_IF;*)
(* -----------------------------------------------------------------------------*)

IF IP_C.TIME_RESET THEN (* Alle Timer ruecksetzen *)
	IP_C.TIME_RESET := FALSE; (* Reset rücksetzen *)
	c_time := tx; (* Connect Timer ruecksetzen *)
	s_time := tx; (* Send Timer ruecksetzen *)
	r_time := tx; (* Receive Timer ruecksetzen *)

	c_status := BYTE#0; (* letzten Connect Fehler rücksetzen *)
	s_status := BYTE#0; (* letzten Send Fehler rücksetzen *)
	r_status := BYTE#0; (* letzten Receive Fehler rücksetzen *)
END_IF;

(* ---------------------------------------------- *)

CASE state OF

UDP_INIT: (* UDP_CLIENT + SERVER *)
	socket := SysSockCreate(SOCKET_AF_INET, SOCKET_DGRAM, SOCKET_IPPROTO_IP);
	IF socket < 0 THEN
		c_status := 1; (* SysSockCreate failed *)
		state := C_CLOSE;
	ELSE
		SysSockSetOption(socket, SOCKET_SOL, SOCKET_SO_BROADCAST, ADR(dint_true), SIZEOF(dint_true)); (* allow broadcast *)
		SysSockIoctl(socket, SOCKET_FIONBIO, ADR(dint_true)); (* put socket in non-blocking mode *)
		sockaddr.sin_family := SOCKET_AF_INET;
		sockaddr.sin_port := SysSockHtons(c_port);
		sockaddr.sin_addr := SEL(c_mode = 1, SOCKET_INADDR_ANY, SysSockNtohl(c_ip));

		IF c_mode >= 2 THEN (* SERVER Mode *)
			IF SysSockBind(socket, ADR(sockaddr), SIZEOF(sockaddr)) THEN
				c_ready := TRUE; (* Connected *)
				state:= C_WAIT;
			ELSE
				c_status := 2; (* SysSockBind failed *)
				state := C_CLOSE;
			END_IF;
		ELSE
			c_ready := TRUE; (* Connected *)
			state:= C_WAIT;
		END_IF;
	END_IF;

(* ---------------------------------------------- *)

TC_INIT: (* TCP-CLIENT (AKTIV) *)
	socket := SysSockCreate(SOCKET_AF_INET, SOCKET_STREAM, SOCKET_IPPROTO_IP);
	IF socket < 0 THEN
		c_status := 1;  (* SysSockCreate failed *)
		state := C_CLOSE;
	ELSE
		IF plc_841 OR plc_881 THEN
			SysSockSetOption(socket,6,SOCKET_TCP_NODELAY, ADR(dint_true), SIZEOF(dint_true)); (* Set Push-Bit *)
		END_IF;
		SysSockIoctl(socket, SOCKET_FIONBIO, ADR(dint_true)); (* NonBlocking mode *)
		sockaddr.sin_family := SOCKET_AF_INET;
		sockaddr.sin_port := SysSockNtohs(c_port);
		sockaddr.sin_addr := SysSockNtohl(c_ip);
		c_select := FALSE;
		state := TC_CONNECT;
	END_IF;

(* ---------------------------------------------- *)

TC_CONNECT:
	IF NOT c_enable OR c_status = 255 THEN (* keine freigabe oder connect timeout *)
			state:= C_CLOSE;
	ELSE
		IF c_select = FALSE THEN
			IF SysSockConnect(socket,ADR(sockaddr),SIZEOF(sockaddr)) THEN
				c_ready := TRUE; (* Connected *)
				state:= C_WAIT;
			ELSE
				(* Connect durchgeführt, aber noch nicht verbunden, dann optional mit select-abfrage weitermachen *)
				c_select := SYSLIBSOCKETS_OPTION.0; (* Bit 0 = TCP-Client - use SysSockselect *)
			END_IF;
		ELSE
			c_Timeout.tv_sec := 0;
			c_Timeout.tv_usec := 0;
			c_fdWrite.fd_count := 1;
			c_fdWrite.fd_array[0] := socket;
			IF SysSockSelect(SOCKET_FD_SETSIZE,0,ADR(c_fdWrite),0, ADR(c_Timeout)) > 0 THEN
				c_ready := TRUE; (* Connected *)
				state:= C_WAIT;
			END_IF;
		END_IF;
	END_IF;

(* ---------------------------------------------- *)

TS_INIT: (* TCP-SERVER (PASSIV) *)
	server_socket := SysSockCreate(SOCKET_AF_INET, SOCKET_STREAM, SOCKET_IPPROTO_IP); (* Create Socket *)
	IF server_socket = SOCKET_INVALID THEN
		c_status := 1; (* SysSockCreate failed *)
		state:= C_CLOSE;
	ELSE (* Address bindings *)
		SysSockSetOption( server_socket, SOCKET_SOL, SOCKET_SO_REUSEADDR, ADR(dint_true), SIZEOF(dint_true) );
		sockaddr.sin_family:= SOCKET_AF_INET;
		sockaddr.sin_port := SysSockHtons(c_port);
		sockaddr.sin_addr := SOCKET_INADDR_ANY;
		IF NOT SysSockBind(server_socket, ADR(sockaddr), SIZEOF(sockaddr)) THEN
			c_status := 2; (* SysSockBind failed *)
			state := C_CLOSE;
		ELSIF NOT SysSockListen(server_socket, 1) THEN (* erzeugt Warteschlange für eine Verbindung *)
			c_status := 3; (* SysSockListen failed *)
			state:= C_CLOSE;
		ELSE
			SysSockIoctl(server_socket, SOCKET_FIONBIO, ADR(dint_true)); (* NonBlocking mode *)
			state:= TS_OPEN;
		END_IF;
	END_IF;

(* ---------------------------------------------- *)

TS_OPEN: (* Waiting for incomming connection *)
	sockaddr_size := SIZEOF(sockaddr);
	socket := SysSockAccept(server_socket, ADR(sockaddr), ADR(sockaddr_size));

	IF socket <> SOCKET_INVALID THEN (* neuer Verbindungswunsch vorhanden *)
		IF c_mode = BYTE#2 AND sockaddr.sin_addr <> SysSockNtohl(c_ip) THEN (* Mode 2 = TCP + PASSIVE + PORT + IP  auf richtige Partner-IP prüfen *)
			state:= C_CLOSE;
		ELSE
			IF plc_841 OR plc_881 THEN
				SysSockSetOption(socket, 6, SOCKET_TCP_NODELAY, ADR(dint_true), SIZEOF(dint_true)); (* Set Push-Bit *)
			END_IF;
			SysSockIoctl(socket, SOCKET_FIONBIO, ADR(dint_true)); (* NonBlocking mode *)
			c_ready := TRUE; (* Connected *)
			state := C_WAIT;
		END_IF;
	ELSIF NOT c_enable THEN (* keine freigabe mehr ? *)
			state:= C_CLOSE;
	END_IF;

(* ---------------------------------------------- *)

C_WAIT: (* Warten auf Anforderung für Beenden *)
	IF NOT c_enable OR NOT c_ready THEN
		state:= C_CLOSE;
	END_IF

(* ---------------------------------------------- *)

C_CLOSE: (* Close the Sockets *)
	c_ready := FALSE;
	IF socket >= 0 THEN
		IF (NOT plc_841) AND (NOT plc_881) THEN
			SysSockShutdown(socket, 0); (* 870 *)
		END_IF;
		SysSockClose(socket);
		socket := SOCKET_INVALID;
	END_IF
	IF server_socket >= 0 THEN
		IF (NOT plc_841) AND (NOT plc_881) THEN
			SysSockShutdown(server_socket, 0); (* 870 *)
		END_IF;
		SysSockClose(server_socket);
		server_socket := SOCKET_INVALID;
	END_IF
	state:= STOP;
END_CASE;

(* ---------------------------------------------- *)

IF c_ready THEN
	IF NOT c_ready_old THEN (* Verbindung aufgebaut - positive Flanke erkannt *)
		IP_C.C_STATE := 254;
		IP_C.TIME_RESET := TRUE; (* Alle Timer ruecksetzen *)
		(* ---------------------- Debug-Message ----------------------------*)
		(*IF _debug_enable THEN
			LOG_CL.NEW_MSG := 'IP_CON: CONNECTED -IP_ID ~6';
			LOG_CL.PRINTF[6] := INT_TO_STRING(debug_ID);
			LOG_MSG();
		END_IF;*)
		(* -----------------------------------------------------------------------------*)
	ELSE
		IP_C.C_STATE := 255; (* Verbindung ist aufgebaut *)
	END_IF;
ELSE
	IF c_ready_old THEN (* Verbindung abgebaut - negative Flanke erkannt *)
		IP_C.C_STATE := 1;
		IP_C.MAILBOX[1] := 0; (* Receive Info rücksetzen *)
		IP_C.MAILBOX[2] := 0; (* Send-Pause rücksetzen *)
		IP_C.MAILBOX[3] := 0; (* Receive-Pause rücksetzen *)
		IF NOT new_connection THEN
			s_active := FALSE; (* Sendeaktivitäten stoppen *)
			s_req := FALSE; (* Sendefreigabe rücksetzen *)
			S_BUF.SIZE := 0; (* Sendelänge löschen *)
			(* IP_C.TIME_RESET := TRUE; *) (* Alle Timer ruecksetzen *)
		END_IF;
		(* ---------------------- Debug-Message ----------------------------*)
		(*IF _debug_enable THEN
			LOG_CL.NEW_MSG := 'IP_CON: DISCONNECTED';
			LOG_MSG();
		END_IF;*)
		(* -----------------------------------------------------------------------------*)
	ELSE
		IP_C.C_STATE := 0; (* Verbindung ist abgebaut *)
	END_IF;
END_IF;

c_ready_old := c_ready;

(* Der Datenempfang wird angehalten solange ein Sendevorgang läuft *)
(* sonst kann es vorkommen das die Antwort-daten schon empfangen werden, *)
(* bevor der Sendevorgang vom programm abgeschlossen wurde *)

IF c_ready AND NOT s_active AND IP_C.MAILBOX[3] = 0 THEN
	IF R_BUF.SIZE >= INT_TO_UINT(r_max_size) THEN
		R_BUF.SIZE := UINT#0;
		r_status := 254; (* Empfangsbuffer wegen Überlauf rückgesetzt *)
	END_IF;

	r_offset := SEL(udp_mode,UINT_TO_INT(R_BUF.SIZE),0);
	r_count := r_max_size - r_offset;

	IF udp_mode THEN
		bytes_received := SysSockRecvFrom(socket, ADR(R_BUF.BUFFER), r_count, 0, ADR(sockaddr), SIZEOF(sockaddr));

		IF c_mode = BYTE#3 AND sockaddr.sin_addr <> SysSockNtohl(c_ip) THEN (* Mode 3 = UDP + PASSIVE + PORT + IP  auf richtige Partner-IP prüfen *)
			bytes_received := 0;
			R_BUF.SIZE := UINT#0;
			sockaddr.sin_port := SysSockNtohs(c_port);
			sockaddr.sin_addr := SysSockNtohl(c_ip);
		END_IF;

	ELSE
		bytes_received := SysSockRecv(socket, ADR(R_BUF.BUFFER[r_offset]), r_count, 0);
	END_IF;

	(*UDP: IPC returns -1 if no data available or error occured,841 returns -1 if error occured and 0 if no data available*)
	CASE bytes_received OF
	-2147483648..-1: ; (* No data available or error occured *)
	 0: IF NOT udp_mode THEN (* TCP-Mode: socket wurde von remote geschlossen *)
			c_status := 253;
			c_ready := FALSE;
		END_IF;
	ELSE (* daten wurden empfangen *)
  		r_time := tx; (* Receive Timer ruecksetzen *)
		R_BUF.SIZE := INT_TO_UINT(r_offset + DINT_TO_UINT(bytes_received)); (* aktuelle buffersize eintragen *)
		IP_C.MAILBOX[1] := IP_C.MAILBOX[1] + 1; (* Receive Info *)
		IF IP_C.MAILBOX[1] = 0 THEN IP_C.MAILBOX[1] := 1; END_IF;

		(* ---------------------- Debug-Message ----------------------------*)
		(*IF _debug_enable THEN
			LOG_CL.NEW_MSG := 'IP_REC DATA: POS: ~1 : SIZE: ~2 TOTAL ~3 -IP_ID ~6';
			LOG_CL.PRINTF[1] := INT_TO_STRING(r_offset);
			LOG_CL.PRINTF[2] := INT_TO_STRING(r_count);
			LOG_CL.PRINTF[3] := UINT_TO_STRING(R_BUF.SIZE);
			LOG_CL.PRINTF[6] := INT_TO_STRING(debug_ID);
			LOG_MSG();
		END_IF;*)
		(* -----------------------------------------------------------------------------*)

	END_CASE
END_IF;

(* ---------------------------------------------- *)

IF S_BUF.SIZE > 0 THEN
	IF c_ready AND c_enable THEN
		IF NOT s_active AND IP_C.MAILBOX[2] = 0 THEN
			(* Gesamtanzahl an Bytes limitieren und uebergeben *)
			s_total := LIMIT(0,UINT_TO_INT(S_BUF.SIZE),r_max_size);
			s_cur_pos  := 0;
			s_cur_size := 0;
			s_start := TRUE; (* Daten kopieren und senden anstossen *)
			s_active := TRUE; (* Sende-Betrieb aktivieren *)
			(* ---------------------- Debug-Message ----------------------------*)
			(*IF _debug_enable THEN
				LOG_CL.NEW_MSG := 'IP_SEN INIT: TOTAL: ~1 -IP_ID ~6';
				LOG_CL.PRINTF[1] := INT_TO_STRING(S_TOTAL);
				LOG_CL.PRINTF[6] := INT_TO_STRING(debug_ID);
				LOG_MSG();
			END_IF;*)
			(* -----------------------------------------------------------------------------*)
		END_IF;

		IF s_done OR s_start THEN (* Daten senden aktiv *)

			s_start := FALSE;
			s_cur_pos := s_cur_pos + s_cur_size; (* neue Sende-Datenposition bestimmen *)
			IF s_total > s_cur_pos THEN (* weitere Daten zum senden vorhanden ? *)
				s_cur_size := s_total - s_cur_pos;
				s_cur_size := LIMIT(0, s_cur_size, s_max_size); (* Telegrammlänge begrenzen *)

				(* ---------------------- Debug-Message ----------------------------*)
				(*IF _debug_enable THEN
					LOG_CL.NEW_MSG := 'IP_SEN DATA: POS: ~1 : SIZE: ~2 TOTAL ~3 -IP_ID ~6';
					LOG_CL.PRINTF[1] := INT_TO_STRING(S_CUR_POS);
					LOG_CL.PRINTF[2] := INT_TO_STRING(S_CUR_SIZE);
					LOG_CL.PRINTF[3] := INT_TO_STRING(S_TOTAL);
					LOG_CL.PRINTF[6] := INT_TO_STRING(debug_ID);
					LOG_MSG();
				END_IF;*)
				(* -----------------------------------------------------------------------------*)

				s_time := tx; (* Send Timer ruecksetzen *)
				r_time := tx; (* Receive Timer ruecksetzen *)
				s_req := TRUE;

			ELSE
				(* keine weitere Sendedaten vorhanden -> Senden beenden *)
				s_req := FALSE;
				s_active := FALSE;
				S_BUF.SIZE := 0;
				(* ---------------------- Debug-Message ----------------------------*)
				(*IF _debug_enable THEN
					LOG_CL.NEW_MSG := 'IP_SEN FINISH -IP_ID ~6';
					LOG_CL.PRINTF[6] := INT_TO_STRING(debug_ID);
					LOG_MSG();
				END_IF;*)
				(* -----------------------------------------------------------------------------*)
			END_IF;
		END_IF;
	END_IF;
END_IF;

IF s_req THEN
	s_done := FALSE;
	IF udp_mode THEN
		bytes_sent := SysSockSendTo(socket, ADR(S_BUF.BUFFER[s_cur_pos]), s_cur_size, 0, ADR(sockaddr), SIZEOF(sockaddr));
	ELSE
		bytes_sent := SysSockSend(socket, ADR(S_BUF.BUFFER[s_cur_pos]), s_cur_size, 0);
	END_IF;

	CASE bytes_sent OF
	-2147483648..-1:	; (* ERROR: Noch nicht bereit um Daten aufzunehmen -> nächsten Zyklus wieder probieren *)
	 0: IF NOT udp_mode THEN (* TCP-Mode: socket wurde von remote geschlossen *)
			c_status := 253;
			c_ready := FALSE;
		END_IF;
	ELSE
		s_done := TRUE;
		s_cur_size := DINT_TO_INT(bytes_sent); (* Anzahl der wirklich versendeten Bytes übernehmen *)
		(* ---------------------- Debug-Message ----------------------------*)
		(*IF _debug_enable THEN
			LOG_CL.NEW_MSG := 'IP_SEN SEND_COUNT ~1 -IP_ID ~6';
			LOG_CL.PRINTF[1] := DINT_TO_STRING(s_cur_size);
			LOG_CL.PRINTF[6] := INT_TO_STRING(debug_ID);
			LOG_MSG();
		END_IF;*)
		(* -----------------------------------------------------------------------------*)
	END_CASE
END_IF;

(* ---------------------------------------------- *)

IF IP_C.R_OBSERVE = FALSE OR s_active THEN
    r_time := tx;
END_IF;

IF c_status = 0 AND tx - c_time > error_time AND c_enable AND NOT c_ready AND c_mode < 2 THEN (* Connect Timeout *)
	c_status := 255; (* Timeout-Fehler ausgeben *)
END_IF;
IF s_status = 0 AND tx - s_time > error_time AND s_active THEN (* Send Timeout *)
	s_status := 255; (* Timeout-Fehler ausgeben *)
END_IF;
IF r_status = 0 AND tx - r_time > error_time AND c_ready AND IP_C.R_OBSERVE THEN (* Receive Timeout *)
	r_status := 255; (* Timeout-Fehler ausgeben *)
END_IF;

IP_C.ERROR := OSCAT_BASIC.DWORD_OF_BYTE(c_status,s_status,r_status,0);

(* ---------------------- Debug-Message ----------------------------*)
(*IF  _debug_enable THEN
	IF (IP_C.ERROR <> debug_lasterror) THEN
		LOG_CL.NEW_MSG := 'IP_ERROR ~1 -IP_ID ~6';
		LOG_CL.PRINTF[1] := DWORD_TO_STRING(IP_C.ERROR);
		LOG_CL.PRINTF[6] := INT_TO_STRING(debug_ID);
		LOG_MSG();

		debug_lasterror := IP_C.ERROR;
		debug_last_id := debug_ID;
	END_IF;
END_IF;*)
(* -----------------------------------------------------------------------------*)

(* revision history
ks	18. oct. 2008	rev 1.0
	original version
ks	05. jan. 2009	rev 1.1
	zusätzlichen Parameter "Port" hinzugefügt, und Code bei Verbindungsaufbau angepasst
ks	28. feb. 2009	rev 1.2
	connect code angepasst und verkürzung der zyklen bei Send
ks	20. oct. 2009	rev 1.3
	network_buffer basis 0
ks	06. dec. 2009	rev 1.4
	receive_count MAILBOX[1]
ks	10. nov. 2010	rev 1.5
	send_pause MAILBOX[2] and receive_pause MAILBOX[3] 
ks	07. feb. 2011	rev 1.6
	Fehlercode 253 bei Remote-Verbindungsabbruch 
ks	30. may. 2011	rev 1.7
	Fehler bei Empfangsüberwachung
ks	26. july. 2011	rev 1.8
	Error-Reset, diverse optimierungen 
ks	26. feb. 2012	rev 1.9
	Code-Optimierung für höhere kompatibilität
*)

END_FUNCTION_BLOCK

// POUs/DRIVER/IRTRANS_DECODE
FUNCTION_BLOCK IRTRANS_DECODE
VAR_IN_OUT
	IP_C : IP_C; (* IP_Control Verwaltungsstruktur *)
	R_BUF : NETWORK_BUFFER_SHORT;
END_VAR
VAR_OUTPUT
	CMD : BOOL;
	DEV : STRING;
	KEY : STRING;
	ERROR : BOOL;
END_VAR
VAR
	i : INT;
	stop : INT;
	pt : POINTER TO BYTE;
	buffer : POINTER TO ARRAY[0..32000] OF BYTE;
	size : UINT;
	z : BYTE;
END_VAR

(*

version 1.2		06. dec. 2009
programmer 		ks
tested by		ks

*)

size := R_BUF.SIZE;

(* do nothing if the buffer is empty *)
IF size > 0 AND IP_C.MAILBOX[1] <> z THEN
	i := 0;
	error := TRUE;
	stop := size - 2;
	(* read characters before first comma and store in device *)
	pt := ADR(dev);
	buffer := ADR(R_BUF.BUFFER);
	WHILE i < stop DO
		IF buffer^[i] = 44 THEN EXIT; END_IF;
		pt^ := buffer^[i];
		pt := pt + 1;
		i := i + 1;
	END_WHILE;
	(* terminate the device string *)
	pt^ := 0;
	(* read after first comma and store in key *)
	i := i + 1;
	pt := ADR(key);
	WHILE i < stop DO
		pt^ := buffer^[i];
		pt := pt + 1;
		i := i + 1;
	END_WHILE;
	(* terminate the key string *)
	pt^:= 0;
	(* check if last two characters are $R$N 13, 10 *)
	IF buffer^[i] <> 13 AND buffer^[i+1] <> 10 THEN	RETURN;	END_IF;
	(* check if device and key are present *)
	IF LEN(dev) = 0 OR LEN(key) = 0 THEN RETURN; END_IF;
	(* a valid transmission has been received *)
	cmd := TRUE;
	error := FALSE;
ELSE
	error := FALSE;
	cmd := FALSE;
END_IF;

z := IP_C.MAILBOX[1];

(* revision history
ks	18. oct. 2008	rev 1.0
	original version
ks	20. oct. 2009	rev 1.1
	Networkbuffer und Buffer-funktionen auf Basis 0
ks	06. dec. 2009	rev 1.2
	Codeanpassung für IRTRANS_SERVER
*)

END_FUNCTION_BLOCK

// POUs/DRIVER/IRTRANS_SERVER
FUNCTION_BLOCK IRTRANS_SERVER
VAR_IN_OUT
	IP_C : IP_C; (* IP_Control Verwaltungsstruktur *)
	S_BUF : NETWORK_BUFFER_SHORT;
	R_BUF : NETWORK_BUFFER_SHORT;
END_VAR
VAR_INPUT
	UDP_TCP : BOOL;
END_VAR
VAR_OUTPUT
	S_ENABLE : BOOL;
	R_ENABLE : BOOL;
	ERROR : DWORD;
END_VAR
VAR
	t : TON;
END_VAR

(*
version 1.1		17. may. 2011
programmer 		ks
tested by			ks
*)

IF NOT IP_C.C_ENABLE THEN
	(* IP Datenverkehr einrichten *)
	IP_C.C_PORT := WORD#0; (* Portnummer eintragen *)
	IP_C.C_IP := DWORD#00; (* IP eintragen *)
	IP_C.C_MODE := SEL(UDP_TCP,5,4); (* 4 = Mode: TCP+PASSIV+PORT / 5 = Mode: UDP+PASSIV+PORT*)
	IP_C.C_ENABLE := TRUE; (* Verbindungsaufbau freigeben *)
	IP_C.R_OBSERVE := FALSE; (* Datenempfang ueberwachen *)
	IP_C.TIME_RESET := TRUE; (* Zeitueberwachung rücksetzen *)
	S_BUF.SIZE := UINT#0; (* Sendedaten rücksetzen *)
	R_BUF.SIZE := UINT#0; (* Empfangsdaten rücksetzen *)
END_IF;

R_ENABLE := IP_C.C_STATE > 127;
S_ENABLE := R_ENABLE AND (IP_C.MAILBOX[1] > 0 OR IP_C.C_MODE <> 5);
ERROR := IP_C.ERROR;

t(IN:= IP_C.ERROR > 0, PT:=T#5s);
IF t.Q THEN
	IP_C.TIME_RESET := TRUE; (* Error Reset *)
END_IF;

(* revision history
ks	6. dec 2009		rev 1.0
	original version

ks	17. may 2011		rev 1.1
	neue Fehlerausgabe und Empfangsbuffer rücksetzen
*)

END_FUNCTION_BLOCK

// POUs/DRIVER/IRTRANS_RCV_1
FUNCTION_BLOCK IRTRANS_RCV_1
VAR_INPUT CONSTANT
	DEV_CODE : STRING;
	KEY_CODE : STRING;
END_VAR
VAR_INPUT
	CMD : BOOL;
END_VAR
VAR_IN_OUT
	DEV : STRING;
	KEY : STRING;
END_VAR
VAR_OUTPUT
	Q : BOOL;
END_VAR


(*

version 1.3	06. dec. 2009
programmer 	hugo
tested by		oscat

*)

Q := cmd AND dev_code = dev AND key_code = key;

(* revision history
hm	2. jan 2008		rev 1.0
	original version

hm	20. 6. 2008		rev 1.1
	performance improvement

hm	19. oct. 2008	rev 1.2
	changed input device_code to dev_code and device to dev for compatibility reasons

hm	06. dec. 2008	rev 1.3
	IRTRANS_1 renamed to IRTRANS_RCV_1

*)

END_FUNCTION_BLOCK

// POUs/DRIVER/IRTRANS_RCV_4
FUNCTION_BLOCK IRTRANS_RCV_4
VAR_INPUT CONSTANT
	DEV_CODE : STRING;
	KEY_CODE_0 : STRING;
	KEY_CODE_1 : STRING;
	KEY_CODE_2 : STRING;
	KEY_CODE_3 : STRING;
END_VAR
VAR_INPUT
	CMD : BOOL;
END_VAR
VAR_IN_OUT
	DEV : STRING;
	KEY : STRING;
END_VAR
VAR_OUTPUT
	Q0, Q1, Q2, Q3 : BOOL;
END_VAR
VAR_TEMP
	decode: BOOL;
END_VAR

(*

version 1.3	06. dec. 2009
programmer 	hugo
tested BY	oscat

*)

decode := cmd AND dev_code = dev;

Q0 := key = key_code_0 AND decode;
Q1 := key = key_code_1 AND decode;
Q2 := key = key_code_2 AND decode;
Q3 := key = key_code_3 AND decode;



(* revision history
hm	2. jan 2008		rev 1.0
	original version

hm	17. oct. 2008	rev 1.1
	improved performance

hm	19. oct. 2008	rev 1.2
	changed input device_code to dev_code and device to dev for compatibility reasons

hm	06. dec. 2008	rev 1.3
	IRTRANS_1 renamed to IRTRANS_RCV_4

*)

END_FUNCTION_BLOCK

// POUs/DRIVER/IRTRANS_RCV_8
FUNCTION_BLOCK IRTRANS_RCV_8
VAR_INPUT CONSTANT
	dev_code : STRING;
	key_code_0 : STRING;
	key_code_1 : STRING;
	key_code_2 : STRING;
	key_code_3 : STRING;
	key_code_4 : STRING;
	key_code_5 : STRING;
	key_code_6 : STRING;
	key_code_7 : STRING;
END_VAR
VAR_INPUT
	CMD : BOOL;
END_VAR
VAR_IN_OUT
	DEV : STRING;
	KEY : STRING;
END_VAR
VAR_OUTPUT
	Q0, Q1, Q2, Q3, Q4, Q5, Q6, Q7 : BOOL;
END_VAR
VAR_TEMP
	decode: BOOL;
END_VAR

(*

version 1.3	06. dec. 2009
programmer 	hugo
tested BY	oscat

*)

decode := cmd AND dev_code = dev;

Q0 := key = key_code_0 AND decode;
Q1 := key = key_code_1 AND decode;
Q2 := key = key_code_2 AND decode;
Q3 := key = key_code_3 AND decode;
Q4 := key = key_code_4 AND decode;
Q5 := key = key_code_5 AND decode;
Q6 := key = key_code_6 AND decode;
Q7 := key = key_code_7 AND decode;


(* revision history
hm	2. jan 2008		rev 1.0
	original version

hm	17. oct 2008	rev 1.1
	improved performance

hm	19. oct. 2008	rev 1.2
	changed input device_code to dev_code and device to dev for compatibility reasons

hm	06. dec. 2008	rev 1.3
	IRTRANS_1 renamed to IRTRANS_RCV_8

*)

END_FUNCTION_BLOCK

// POUs/DRIVER/IRTRANS_SND_1
FUNCTION_BLOCK IRTRANS_SND_1
VAR_INPUT CONSTANT
	DEV_CODE : STRING;
	KEY_CODE : STRING;
END_VAR
VAR_INPUT
	IN : BOOL;
	T_REPEAT : TIME;
END_VAR
VAR_IN_OUT
	IP_C : IP_C; (* IP_Control Verwaltungsstruktur *)
	S_BUF : NETWORK_BUFFER_SHORT;
END_VAR
VAR_OUTPUT
	KEY : BYTE;
END_VAR
VAR
	skey : STRING;
	size : INT;
	str : STRING;
	t : TON;
	k : BYTE;
	lk : BYTE;
	d : BOOL;
END_VAR

(*
version 1.0		06. dec. 2009
programmer 		ks
tested by		ks
*)

d := IP_C.C_STATE > 127 AND (IP_C.MAILBOX[1] > 0 OR IP_C.C_MODE <> 5);
IF NOT d THEN RETURN; END_IF;

t(IN:= lk = k , PT:=T_REPEAT);

IF S_BUF.SIZE = 0 THEN
	IF IN THEN
		skey := KEY_CODE; k := 1;
	ELSE
		lk := 0;
		KEY := 0;
		RETURN; (* beenden wenn kein Key aktiv *)
	END_IF;

	IF lk <> k OR T.Q THEN (* anderer Key oder repeat wartezeit abgelaufen *)
		str := CONCAT('snd ',dev_code);
		str := CONCAT(str,',');
		str := CONCAT(str,skey);
		size := LEN(str);
		OSCAT_BASIC._STRING_TO_BUFFER(STR:=str, POS:=0, PT:=ADR(S_BUF.BUFFER), SIZE:=size);
		S_BUF.SIZE := size; (* Sendelänge eintragen *)
		KEY := k;
		lk := k; (* letzten Key speichern *)
		t(IN:=FALSE); (* Reset Time *)
	END_IF;
END_IF;

(* revision history
hm	6. dec 2009		rev 1.0
	original version
*)

END_FUNCTION_BLOCK

// POUs/DRIVER/IRTRANS_SND_4
FUNCTION_BLOCK IRTRANS_SND_4
VAR_INPUT CONSTANT
	DEV_CODE : STRING;
	KEY_CODE_0 : STRING;
	KEY_CODE_1 : STRING;
	KEY_CODE_2 : STRING;
	KEY_CODE_3 : STRING;
END_VAR
VAR_INPUT
	IN_0 : BOOL;
	IN_1 : BOOL;
	IN_2 : BOOL;
	IN_3 : BOOL;
	T_REPEAT : TIME;
END_VAR
VAR_IN_OUT
	IP_C : IP_C; (* IP_Control Verwaltungsstruktur *)
	S_BUF : NETWORK_BUFFER_SHORT;
END_VAR
VAR_OUTPUT
	KEY : BYTE;
END_VAR
VAR
	skey : STRING;
	size : INT;
	str : STRING;
	t : TON;
	k : BYTE;
	lk : BYTE;
	d : BOOL;
END_VAR

(*
version 1.0		06. dec. 2009
programmer 		ks
tested by		ks
*)

d := IP_C.C_STATE > 127 AND (IP_C.MAILBOX[1] > 0 OR IP_C.C_MODE <> 5);
IF NOT d THEN RETURN; END_IF;

t(IN:= lk = k , PT:=T_REPEAT);

IF S_BUF.SIZE = 0 THEN
	IF IN_0 THEN
		skey := KEY_CODE_0; k := 1;
	ELSIF IN_1 THEN
		skey := KEY_CODE_1; k := 2;
	ELSIF IN_2 THEN
		skey := KEY_CODE_2; k := 3;
	ELSIF IN_3 THEN
		skey := KEY_CODE_3; k := 4;
	ELSE
		lk := 0;
		KEY := 0;
		RETURN; (* beenden wenn kein Key aktiv *)
	END_IF;

	IF lk <> k OR T.Q THEN (* anderer Key oder repeat wartezeit abgelaufen *)
		str := CONCAT('snd ',dev_code);
		str := CONCAT(str,',');
		str := CONCAT(str,skey);
		size := LEN(str);
		OSCAT_BASIC._STRING_TO_BUFFER(STR:=str, POS:=0, PT:=ADR(S_BUF.BUFFER), SIZE:=size);
		S_BUF.SIZE := size; (* Sendelänge eintragen *)
		KEY := k;
		lk := k; (* letzten Key speichern *)
		t(IN:=FALSE); (* Reset Time *)
	END_IF;
END_IF;

(* revision history
hm	6. dec 2009		rev 1.0
	original version
*)

END_FUNCTION_BLOCK

// POUs/DRIVER/IRTRANS_SND_8
FUNCTION_BLOCK IRTRANS_SND_8
VAR_INPUT CONSTANT
	DEV_CODE : STRING;
	KEY_CODE_0 : STRING;
	KEY_CODE_1 : STRING;
	KEY_CODE_2 : STRING;
	KEY_CODE_3 : STRING;
	KEY_CODE_4 : STRING;
	KEY_CODE_5 : STRING;
	KEY_CODE_6 : STRING;
	KEY_CODE_7 : STRING;
END_VAR
VAR_INPUT
	IN_0 : BOOL;
	IN_1 : BOOL;
	IN_2 : BOOL;
	IN_3 : BOOL;
	IN_4 : BOOL;
	IN_5 : BOOL;
	IN_6 : BOOL;
	IN_7 : BOOL;
	T_REPEAT : TIME;
END_VAR
VAR_IN_OUT
	IP_C : IP_C; (* IP_Control Verwaltungsstruktur *)
	S_BUF : NETWORK_BUFFER_SHORT;
END_VAR
VAR_OUTPUT
	KEY : BYTE;
END_VAR
VAR
	skey : STRING;
	size : INT;
	str : STRING;
	t : TON;
	k : BYTE;
	lk : BYTE;
	d : BOOL;
END_VAR

(*
version 1.0		06. dec. 2009
programmer 		ks
tested by		ks
*)

d := IP_C.C_STATE > 127 AND (IP_C.MAILBOX[1] > 0 OR IP_C.C_MODE <> 5);
IF NOT d THEN RETURN; END_IF;

t(IN:= lk = k , PT:=T_REPEAT);

IF S_BUF.SIZE = 0 THEN
	IF IN_0 THEN
		skey := KEY_CODE_0; k := 1;
	ELSIF IN_1 THEN
		skey := KEY_CODE_1; k := 2;
	ELSIF IN_2 THEN
		skey := KEY_CODE_2; k := 3;
	ELSIF IN_3 THEN
		skey := KEY_CODE_3; k := 4;
	ELSIF IN_4 THEN
		skey := KEY_CODE_4; k := 5;
	ELSIF IN_5 THEN
		skey := KEY_CODE_5; k := 6;
	ELSIF IN_6 THEN
		skey := KEY_CODE_6; k := 7;
	ELSIF IN_7 THEN
		skey := KEY_CODE_7; k := 8;
	ELSE
		lk := 0;
		KEY := 0;
		RETURN; (* beenden wenn kein Key aktiv *)
	END_IF;

	IF lk <> k OR T.Q THEN (* anderer Key oder repeat wartezeit abgelaufen *)
		str := CONCAT('snd ',dev_code);
		str := CONCAT(str,',');
		str := CONCAT(str,skey);
		size := LEN(str);
		OSCAT_BASIC._STRING_TO_BUFFER(STR:=str, POS:=0, PT:=ADR(S_BUF.BUFFER), SIZE:=size);
		S_BUF.SIZE := size; (* Sendelänge eintragen *)
		KEY := k;
		lk := k; (* letzten Key speichern *)
		t(IN:=FALSE); (* Reset Time *)
	END_IF;
END_IF;

(* revision history
hm	6. dec 2009		rev 1.0
	original version
*)

END_FUNCTION_BLOCK

// POUs/CONVERT/IS_IP4
FUNCTION IS_IP4 : BOOL
VAR_INPUT
	str : STRING;
END_VAR


(*
version 1.1	10. mar 2009
programmer 	kurt
tested by		hugo

IS_IP4 testet ob ein string eine gültige IPv4 Adresse enthält.

*)

IS_IP4 := OSCAT_BASIC.COUNT_CHAR(str, 46) = 3;


(* revision history
hm	1. mar. 2008	rev 1.0
	original version

hm	10. mar. 2009	rev 1.1
	new code

*)

END_FUNCTION

// POUs/CONVERT/IS_URLCHR
FUNCTION IS_URLCHR : BOOL
VAR_INPUT
	IN : BYTE;
END_VAR


(*
version 1.0		27. apr. 2008
programmer 		hugo
tested by		hugo

IS_URL_CHR is true if a string contains only non reserved characters for an url.
the non reserved characters are : [A..Z], [a..z], [0..9], -_.~

*)

IS_URLCHR := ((IN > 47) AND (IN < 58)) OR ((IN > 64) AND (IN < 91)) OR ((IN > 96) AND (IN < 123)) OR (in = 126) OR (in = 95) OR (in =45) OR (in =46);


(* revision history
hm		27. apr. 2008	rev 1.0
	original version

*)

END_FUNCTION

// POUs/NETWORK/LOG_VIEWPORT
FUNCTION_BLOCK LOG_VIEWPORT
VAR_IN_OUT
	LC : LOG_CONTROL;
	LV : us_LOG_VIEWPORT;
END_VAR
VAR
	pos : INT;
	count : INT;
	idx : INT;
	base : INT;
	update_pos : BOOL;
END_VAR

(*
version 1.1		05 mai 2012
programmer		ks
tested BY		ks

LOG_VIEWPORT erzeugt einen Liste der Meldungen des Loggingbuffers die innerhalb einer virtuellen Ansicht enthalten sind.
*)

(* Scroll Button verarbeiten *)
IF LV.MOVE_TO_X <> 0 THEN
	CASE LV.MOVE_TO_X OF
	30000: pos := 1 ; (* älteste Meldung anzeigen *)
	30001: pos := LC.SIZE; (* neueste Meldung anzeigen *)
	30002: pos := pos + LV.COUNT; (* eine Seite nach unten blättern -> Richtung neuere Nachrichten *)
	30003: pos := pos - LV.COUNT; (* eine Seite nach oben blättern -> Richtung ältere Nachrichten *)
	ELSE
		pos := pos + LV.MOVE_TO_X;
	END_CASE;
	update_pos := TRUE;
	LV.MOVE_TO_X := 0;
END_IF;

IF (LV.UPDATE_COUNT <> LC.UPDATE_COUNT) OR update_pos THEN (* Aktualisierung überwachen *)
	LV.UPDATE := TRUE;
	LV.UPDATE_COUNT := LC.UPDATE_COUNT;
	update_pos := FALSE;

	(* pos prüfen und übernehmen *)
	IF LC.RING_MODE THEN
		pos := LIMIT(1,pos,LC.SIZE - LV.COUNT + 1);
	ELSE
		IF LC.IDX > LV.COUNT THEN
			pos := LIMIT(1,pos,LC.IDX - LV.COUNT + 1);
		ELSE
			pos := 1;
		END_IF;
	END_IF;

	(* idxBasis berechnen *)
	base := LC.IDX - pos - LV.COUNT + 1;
	IF LC.RING_MODE THEN 
		(* Anzeige im Ringpuffermodus *)
		FOR count:= 1 TO LV.COUNT DO
			idx := base + count;
			IF idx < 1 THEN
				idx := idx + LC.SIZE;
			END_IF;
			LV.LINE_ARRAY[count] := idx;
		END_FOR;
	ELSE
		(* Anzeige im Normalmodus *)
		FOR count:= 1 TO LV.COUNT DO
			idx := base + count;
			IF idx < 1 THEN
				(* Leere Zeile ausgeben *)
				LV.LINE_ARRAY[count] := 0;
			ELSE
				LV.LINE_ARRAY[count] := idx;
			END_IF;
		END_FOR;
	END_IF;
END_IF;

(* revision history
ks	01. mai 2010	rev 1.0
	original version

ks	05. mai 2012	rev 1.1
	Fehler im Ringmodus

*)

END_FUNCTION_BLOCK

// POUs/NETWORK/MB_CLIENT
FUNCTION_BLOCK MB_CLIENT
VAR_IN_OUT
	IP_C : IP_C;
	S_BUF : NETWORK_BUFFER_SHORT;
	R_BUF : NETWORK_BUFFER_SHORT;
	DATA : ARRAY [0..255] OF WORD;
END_VAR
VAR_INPUT
	DATA_SIZE : INT;
	ENABLE : BOOL;
	UDP : BOOL;
	FC : INT;
	UNIT_ID : BYTE;
	R_ADDR : INT;
	R_POINTS : INT;
	R_DATA_ADR : INT;
	R_DATA_BITPOS : INT;
	W_ADDR : INT;
	W_POINTS : INT;
	W_DATA_ADR : INT;
	W_DATA_BITPOS : INT;
	DELAY : TIME;
END_VAR
VAR_OUTPUT
	ERROR : DWORD;
	BUSY : BOOL;
END_VAR
VAR
	ip_state : BYTE;
	ip_id : BYTE;
	ip_fifo : ip_fifo;
	mask : DWORD;
	w_tmp : WORD;
	idx1 : INT;
	idx2 : INT;
	stop : INT;
	i : INT;
	bit_pos : INT;
	w_mask : WORD;
	b_mask : BYTE;
	count : INT;
	state : INT;
	transaction_id : INT;
	response : INT;
	comp : INT;
	ton_1 : TON;
END_VAR

(*
version 1.2		20. oct. 2009
programmer 		ks
tested BY		ks

MB_CLIENT ermöglicht das Lesen/Schreiben von Daten über das Protokoll Modbus over Ethernet (OpenModbus)
*)

CASE state OF

00: (* Warten auf Delay-Time *)
	TON_1(IN:=ENABLE,PT:=DELAY);

	IF TON_1.Q OR DELAY = T#0s THEN
		TON_1(IN:=FALSE);
		state := 20;
		IP_STATE := BYTE#1; (* Anmelden *)
	END_IF;

20: (* Bei IP_Control anmelden *)
	IF IP_STATE = BYTE#3 THEN
		(* IP Datenverkehr einrichten *)
		IP_C.C_PORT := WORD#0; (* Port von IP_CONTROL verwenden *)
		IP_C.C_IP := DWORD#0; (* IP von IP_CONTROL verwenden *)
		IP_C.C_MODE := BOOL_TO_BYTE(UDP); (* Mode: 0=TCP+ACTIVE+IP , 1=UDP+ACTIVE+IP *)
		IP_C.TIME_RESET := TRUE; (* Zeitueberwachung rücksetzen *)
		IP_C.C_ENABLE := TRUE; (* Verbindungsaufbau freigeben *)
		IP_C.R_OBSERVE := TRUE; (* Empfangsueberwachung *)
		ERROR := DWORD#00; (* letzten Fehler rücksetzen *)

